LIN {X 0,Y 539.068,Z 532.449,A -85,B 0,C 180,E1 4627.318,E2 4627.318} C_VEL
LIN {X 0,Y 539.511,Z 496.056,A -85,B 0,C 180,E1 4628.109,E2 4628.109} C_VEL
LIN {X 0,Y 522.356,Z 463.143,A -85,B 0,C 180,E1 4630.176,E2 4630.176} C_VEL
LIN {X 0,Y 522.421,Z 462.44,A -85,B 0,C 180,E1 4635.931,E2 4635.931} C_VEL
LIN {X 0,Y 522.358,Z 462.44,A -85,B 0,C 180,E1 4641.503,E2 4641.503} C_VEL
LIN {X 0,Y 522.384,Z 462.44,A -85,B 0,C 180,E1 4647.2,E2 4647.2} C_VEL
LIN {X 0,Y 522.47,Z 462.44,A -85,B 0,C 180,E1 4652.377,E2 4652.377} C_VEL
LIN {X 0,Y 522.638,Z 462.44,A -85,B 0,C 180,E1 4657.983,E2 4657.983} C_VEL
LIN {X 0,Y 522.677,Z 462.44,A -85,B 0,C 180,E1 4663.162,E2 4663.162} C_VEL
LIN {X 0,Y 522.728,Z 462.44,A -85,B 0,C 180,E1 4670.012,E2 4670.012} C_VEL
LIN {X 0,Y 522.901,Z 462.44,A -85,B 0,C 180,E1 4675.016,E2 4675.016} C_VEL
LIN {X 0,Y 522.923,Z 462.44,A -85,B 0,C 180,E1 4679.999,E2 4679.999} C_VEL
LIN {X 0,Y 522.848,Z 462.44,A -85,B 0,C 180,E1 4684.982,E2 4684.982} C_VEL
LIN {X 0,Y 522.787,Z 462.44,A -85,B 0,C 180,E1 4690.024,E2 4690.024} C_VEL
LIN {X 0,Y 522.67,Z 462.44,A -85,B 0,C 180,E1 4695.11,E2 4695.11} C_VEL
LIN {X 0,Y 522.589,Z 462.44,A -85,B 0,C 180,E1 4700.342,E2 4700.342} C_VEL
LIN {X 0,Y 522.421,Z 462.44,A -85,B 0,C 180,E1 4706.042,E2 4706.042} C_VEL
LIN {X 0,Y 522.407,Z 462.44,A -85,B 0,C 180,E1 4711.442,E2 4711.442} C_VEL
LIN {X 0,Y 522.38,Z 462.44,A -85,B 0,C 180,E1 4717.488,E2 4717.488} C_VEL
LIN {X 0,Y 522.212,Z 462.44,A -85,B 0,C 180,E1 4723.542,E2 4723.542} C_VEL
LIN {X 0,Y 522.348,Z 462.44,A -85,B 0,C 180,E1 4728.899,E2 4728.899} C_VEL
LIN {X 0,Y 522.594,Z 462.44,A -85,B 0,C 180,E1 4734.992,E2 4734.992} C_VEL
LIN {X 0,Y 535.97,Z 492.125,A -85,B 0,C 180,E1 4736.47,E2 4736.47} C_VEL
LIN {X 0,Y 535.438,Z 535.67,A -85,B 0,C 180,E1 4737.354,E2 4737.354} C_VEL
LIN {X 0,Y 533.837,Z 572.448,A -85,B 0,C 180,E1 4738.666,E2 4738.666} C_VEL
LIN {X 0,Y 531.767,Z 608.408,A -85,B 0,C 180,E1 4740.582,E2 4740.582} C_VEL
LIN {X 0,Y 529.464,Z 642.826,A -85,B 0,C 180,E1 4743.115,E2 4743.115} C_VEL
LIN {X 0,Y 527.341,Z 673.183,A -85,B 0,C 180,E1 4746.073,E2 4746.073} C_VEL
LIN {X 0,Y 525.539,Z 700.097,A -85,B 0,C 180,E1 4749.484,E2 4749.484} C_VEL
LIN {X 0,Y 524.279,Z 723.704,A -85,B 0,C 180,E1 4753.43,E2 4753.43} C_VEL
LIN {X 0,Y 523.54,Z 741.491,A -85,B 0,C 180,E1 4757.473,E2 4757.473} C_VEL
LIN {X 0,Y 523.247,Z 754.217,A -85,B 0,C 180,E1 4761.681,E2 4761.681} C_VEL
LIN {X 0,Y 523.13,Z 760.5,A -85,B 0,C 180,E1 4765.019,E2 4765.019} C_VEL
LIN {X 0,Y 523.088,Z 763.612,A -85,B 0,C 180,E1 4768.341,E2 4768.341} C_VEL
LIN {X 0,Y 523.184,Z 763.555,A -85,B 0,C 180,E1 4771.658,E2 4771.658} C_VEL
LIN {X 0,Y 523.211,Z 759.15,A -85,B 0,C 180,E1 4775.813,E2 4775.813} C_VEL
LIN {X 0,Y 523.34,Z 749.587,A -85,B 0,C 180,E1 4779.997,E2 4779.997} C_VEL
LIN {X 0,Y 523.808,Z 734.142,A -85,B 0,C 180,E1 4784.287,E2 4784.287} C_VEL
LIN {X 0,Y 524.881,Z 712.493,A -85,B 0,C 180,E1 4788.501,E2 4788.501} C_VEL
LIN {X 0,Y 526.437,Z 686.433,A -85,B 0,C 180,E1 4792.268,E2 4792.268} C_VEL
LIN {X 0,Y 528.502,Z 656.362,A -85,B 0,C 180,E1 4795.571,E2 4795.571} C_VEL
LIN {X 0,Y 530.794,Z 623.032,A -85,B 0,C 180,E1 4798.343,E2 4798.343} C_VEL
LIN {X 0,Y 532.941,Z 589.022,A -85,B 0,C 180,E1 4800.442,E2 4800.442} C_VEL
LIN {X 0,Y 534.766,Z 553.339,A -85,B 0,C 180,E1 4802.003,E2 4802.003} C_VEL
LIN {X 0,Y 535.972,Z 516.697,A -85,B 0,C 180,E1 4803.016,E2 4803.016} C_VEL
LIN {X 0,Y 535.534,Z 491.051,A -85,B 0,C 180,E1 4803.488,E2 4803.488} C_VEL
LIN {X 0,Y 522.397,Z 462.44,A -85,B 0,C 180,E1 4805.02,E2 4805.02} C_VEL
LIN {X 0,Y 522.353,Z 462.44,A -85,B 0,C 180,E1 4811.101,E2 4811.101} C_VEL
LIN {X 0,Y 522.357,Z 462.44,A -85,B 0,C 180,E1 4816.441,E2 4816.441} C_VEL
LIN {X 0,Y 522.293,Z 462.44,A -85,B 0,C 180,E1 4822.504,E2 4822.504} C_VEL
LIN {X 0,Y 522.342,Z 462.44,A -85,B 0,C 180,E1 4828.554,E2 4828.554} C_VEL
LIN {X 0,Y 522.502,Z 462.44,A -85,B 0,C 180,E1 4834.24,E2 4834.24} C_VEL
LIN {X 0,Y 522.655,Z 462.44,A -85,B 0,C 180,E1 4839.66,E2 4839.66} C_VEL
LIN {X 0,Y 522.798,Z 462.44,A -85,B 0,C 180,E1 4844.894,E2 4844.894} C_VEL
LIN {X 0,Y 522.789,Z 462.44,A -85,B 0,C 180,E1 4851.23,E2 4851.23} C_VEL
LIN {X 0,Y 523.02,Z 462.44,A -85,B 0,C 180,E1 4856.682,E2 4856.682} C_VEL
LIN {X 0,Y 523.103,Z 462.44,A -85,B 0,C 180,E1 4861.659,E2 4861.659} C_VEL
LIN {X 0,Y 522.951,Z 462.44,A -85,B 0,C 180,E1 4866.651,E2 4866.651} C_VEL
LIN {X 0,Y 522.767,Z 462.44,A -85,B 0,C 180,E1 4871.697,E2 4871.697} C_VEL
LIN {X 0,Y 522.616,Z 462.44,A -85,B 0,C 180,E1 4877.043,E2 4877.043} C_VEL
LIN {X 0,Y 522.614,Z 462.44,A -85,B 0,C 180,E1 4882.124,E2 4882.124} C_VEL
LIN {X 0,Y 522.476,Z 462.44,A -85,B 0,C 180,E1 4887.622,E2 4887.622} C_VEL
LIN {X 0,Y 522.352,Z 462.44,A -85,B 0,C 180,E1 4892.514,E2 4892.514} C_VEL
LIN {X 0,Y 519.895,Z 462.44,A -85,B 0,C 180,E1 4893.928,E2 4893.928} C_VEL
LIN {X 0,Y 514.521,Z 462.44,A -85,B 0,C 180,E1 4896.046,E2 4896.046} C_VEL
LIN {X 0,Y 514.418,Z 462.44,A -85,B 0,C 180,E1 4896.292,E2 4896.292} C_VEL
LIN {X 0,Y 514.484,Z 462.44,A -85,B 0,C 180,E1 4902.629,E2 4902.629} C_VEL
LIN {X 0,Y 514.424,Z 462.947,A -85,B 0,C 180,E1 4909.174,E2 4909.174} C_VEL
LIN {X 0,Y 525.004,Z 483.039,A -85,B 0,C 180,E1 4910.412,E2 4910.412} C_VEL
LIN {X 0,Y 533.703,Z 501.5,A -85,B 0,C 180,E1 4911.496,E2 4911.496} C_VEL
LIN {X 0,Y 532.173,Z 544.934,A -85,B 0,C 180,E1 4912.524,E2 4912.524} C_VEL
LIN {X 0,Y 529.677,Z 588.035,A -85,B 0,C 180,E1 4914.292,E2 4914.292} C_VEL
LIN {X 0,Y 526.477,Z 629.276,A -85,B 0,C 180,E1 4916.773,E2 4916.773} C_VEL
LIN {X 0,Y 523.242,Z 667.514,A -85,B 0,C 180,E1 4919.932,E2 4919.932} C_VEL
LIN {X 0,Y 520.398,Z 700.092,A -85,B 0,C 180,E1 4923.454,E2 4923.454} C_VEL
LIN {X 0,Y 518.057,Z 730.026,A -85,B 0,C 180,E1 4927.669,E2 4927.669} C_VEL
LIN {X 0,Y 516.559,Z 753.744,A -85,B 0,C 180,E1 4932.054,E2 4932.054} C_VEL
LIN {X 0,Y 515.736,Z 772.742,A -85,B 0,C 180,E1 4936.848,E2 4936.848} C_VEL
LIN {X 0,Y 515.308,Z 785.33,A -85,B 0,C 180,E1 4941.552,E2 4941.552} C_VEL
LIN {X 0,Y 515.391,Z 790.904,A -85,B 0,C 180,E1 4944.944,E2 4944.944} C_VEL
LIN {X 0,Y 515.296,Z 793.657,A -85,B 0,C 180,E1 4948.316,E2 4948.316} C_VEL
LIN {X 0,Y 515.217,Z 792.628,A -85,B 0,C 180,E1 4953.37,E2 4953.37} C_VEL
LIN {X 0,Y 515.336,Z 786.917,A -85,B 0,C 180,E1 4957.598,E2 4957.598} C_VEL
LIN {X 0,Y 515.477,Z 776.771,A -85,B 0,C 180,E1 4961.865,E2 4961.865} C_VEL
LIN {X 0,Y 516.124,Z 761.488,A -85,B 0,C 180,E1 4966.182,E2 4966.182} C_VEL
LIN {X 0,Y 517.307,Z 740.375,A -85,B 0,C 180,E1 4970.563,E2 4970.563} C_VEL
LIN {X 0,Y 519.171,Z 714.818,A -85,B 0,C 180,E1 4974.608,E2 4974.608} C_VEL
LIN {X 0,Y 521.784,Z 684.177,A -85,B 0,C 180,E1 4978.371,E2 4978.371} C_VEL
LIN {X 0,Y 524.76,Z 650.107,A -85,B 0,C 180,E1 4981.614,E2 4981.614} C_VEL
LIN {X 0,Y 527.73,Z 614.196,A -85,B 0,C 180,E1 4984.231,E2 4984.231} C_VEL
LIN {X 0,Y 530.638,Z 574.086,A -85,B 0,C 180,E1 4986.362,E2 4986.362} C_VEL
LIN {X 0,Y 532.788,Z 532.447,A -85,B 0,C 180,E1 4987.835,E2 4987.835} C_VEL
LIN {X 0,Y 533.34,Z 499.06,A -85,B 0,C 180,E1 4988.58,E2 4988.58} C_VEL
LIN {X 0,Y 514.575,Z 464.052,A -85,B 0,C 180,E1 4990.795,E2 4990.795} C_VEL
LIN {X 0,Y 514.404,Z 462.44,A -85,B 0,C 180,E1 4990.993,E2 4990.993} C_VEL
LIN {X 0,Y 514.484,Z 462.44,A -85,B 0,C 180,E1 4997.404,E2 4997.404} C_VEL
LIN {X 0,Y 514.46,Z 462.44,A -85,B 0,C 180,E1 5002.622,E2 5002.622} C_VEL
LIN {X 0,Y 514.474,Z 462.44,A -85,B 0,C 180,E1 5008.593,E2 5008.593} C_VEL
LIN {X 0,Y 514.588,Z 462.44,A -85,B 0,C 180,E1 5013.811,E2 5013.811} C_VEL
LIN {X 0,Y 514.737,Z 462.44,A -85,B 0,C 180,E1 5020.271,E2 5020.271} C_VEL
LIN {X 0,Y 514.559,Z 462.44,A -85,B 0,C 180,E1 5026.181,E2 5026.181} C_VEL
LIN {X 0,Y 514.812,Z 462.44,A -85,B 0,C 180,E1 5031.544,E2 5031.544} C_VEL
LIN {X 0,Y 514.985,Z 462.44,A -85,B 0,C 180,E1 5036.628,E2 5036.628} C_VEL
LIN {X 0,Y 514.988,Z 462.44,A -85,B 0,C 180,E1 5041.684,E2 5041.684} C_VEL
LIN {X 0,Y 514.887,Z 462.44,A -85,B 0,C 180,E1 5046.753,E2 5046.753} C_VEL
LIN {X 0,Y 514.784,Z 462.44,A -85,B 0,C 180,E1 5051.879,E2 5051.879} C_VEL
LIN {X 0,Y 514.7,Z 462.44,A -85,B 0,C 180,E1 5057.105,E2 5057.105} C_VEL
LIN {X 0,Y 514.624,Z 462.44,A -85,B 0,C 180,E1 5062.484,E2 5062.484} C_VEL
LIN {X 0,Y 514.455,Z 462.44,A -85,B 0,C 180,E1 5068.089,E2 5068.089} C_VEL
LIN {X 0,Y 514.508,Z 462.44,A -85,B 0,C 180,E1 5073.991,E2 5073.991} C_VEL
LIN {X 0,Y 514.441,Z 462.44,A -85,B 0,C 180,E1 5080.071,E2 5080.071} C_VEL
LIN {X 0,Y 514.235,Z 462.44,A -85,B 0,C 180,E1 5085.036,E2 5085.036} C_VEL
LIN {X 0,Y 514.457,Z 462.44,A -85,B 0,C 180,E1 5089.917,E2 5089.917} C_VEL
LIN {X 0,Y 514.646,Z 462.711,A -85,B 0,C 180,E1 5094.315,E2 5094.315} C_VEL
LIN {X 0,Y 529.385,Z 494.183,A -85,B 0,C 180,E1 5096.03,E2 5096.03} C_VEL
LIN {X 0,Y 528.695,Z 537.141,A -85,B 0,C 180,E1 5096.931,E2 5096.931} C_VEL
LIN {X 0,Y 526.913,Z 574.501,A -85,B 0,C 180,E1 5098.31,E2 5098.31} C_VEL
LIN {X 0,Y 524.661,Z 609.82,A -85,B 0,C 180,E1 5100.243,E2 5100.243} C_VEL
LIN {X 0,Y 522.143,Z 644.081,A -85,B 0,C 180,E1 5102.824,E2 5102.824} C_VEL
LIN {X 0,Y 519.779,Z 675.099,A -85,B 0,C 180,E1 5105.932,E2 5105.932} C_VEL
LIN {X 0,Y 517.806,Z 702.022,A -85,B 0,C 180,E1 5109.458,E2 5109.458} C_VEL
LIN {X 0,Y 516.471,Z 724.789,A -85,B 0,C 180,E1 5113.391,E2 5113.391} C_VEL
LIN {X 0,Y 515.709,Z 741.489,A -85,B 0,C 180,E1 5117.279,E2 5117.279} C_VEL
LIN {X 0,Y 515.361,Z 754.215,A -85,B 0,C 180,E1 5121.553,E2 5121.553} C_VEL
LIN {X 0,Y 515.251,Z 760.499,A -85,B 0,C 180,E1 5124.942,E2 5124.942} C_VEL
LIN {X 0,Y 515.185,Z 763.612,A -85,B 0,C 180,E1 5128.316,E2 5128.316} C_VEL
LIN {X 0,Y 515.201,Z 763.101,A -85,B 0,C 180,E1 5132.437,E2 5132.437} C_VEL
LIN {X 0,Y 515.309,Z 757.598,A -85,B 0,C 180,E1 5136.75,E2 5136.75} C_VEL
LIN {X 0,Y 515.502,Z 748.281,A -85,B 0,C 180,E1 5140.589,E2 5140.589} C_VEL
LIN {X 0,Y 516.085,Z 732.756,A -85,B 0,C 180,E1 5144.82,E2 5144.82} C_VEL
LIN {X 0,Y 517.301,Z 711.169,A -85,B 0,C 180,E1 5149.004,E2 5149.004} C_VEL
LIN {X 0,Y 518.994,Z 685.739,A -85,B 0,C 180,E1 5152.695,E2 5152.695} C_VEL
LIN {X 0,Y 521.168,Z 656.428,A -85,B 0,C 180,E1 5155.951,E2 5155.951} C_VEL
LIN {X 0,Y 523.723,Z 622.883,A -85,B 0,C 180,E1 5158.773,E2 5158.773} C_VEL
LIN {X 0,Y 526.138,Z 587.932,A -85,B 0,C 180,E1 5160.941,E2 5160.941} C_VEL
LIN {X 0,Y 528.053,Z 552.594,A -85,B 0,C 180,E1 5162.487,E2 5162.487} C_VEL
LIN {X 0,Y 529.405,Z 513.93,A -85,B 0,C 180,E1 5163.533,E2 5163.533} C_VEL
LIN {X 0,Y 529.025,Z 493.82,A -85,B 0,C 180,E1 5163.912,E2 5163.912} C_VEL
LIN {X 0,Y 514.476,Z 462.44,A -85,B 0,C 180,E1 5165.67,E2 5165.67} C_VEL
LIN {X 0,Y 514.446,Z 462.44,A -85,B 0,C 180,E1 5170.354,E2 5170.354} C_VEL
LIN {X 0,Y 514.346,Z 462.44,A -85,B 0,C 180,E1 5175.056,E2 5175.056} C_VEL
LIN {X 0,Y 514.413,Z 462.44,A -85,B 0,C 180,E1 5179.933,E2 5179.933} C_VEL
LIN {X 0,Y 514.37,Z 462.44,A -85,B 0,C 180,E1 5185.999,E2 5185.999} C_VEL
LIN {X 0,Y 514.517,Z 462.44,A -85,B 0,C 180,E1 5191.988,E2 5191.988} C_VEL
LIN {X 0,Y 514.658,Z 462.44,A -85,B 0,C 180,E1 5197.518,E2 5197.518} C_VEL
LIN {X 0,Y 514.802,Z 462.44,A -85,B 0,C 180,E1 5202.898,E2 5202.898} C_VEL
LIN {X 0,Y 514.854,Z 462.44,A -85,B 0,C 180,E1 5208.122,E2 5208.122} C_VEL
LIN {X 0,Y 514.886,Z 462.44,A -85,B 0,C 180,E1 5213.247,E2 5213.247} C_VEL
LIN {X 0,Y 514.978,Z 462.44,A -85,B 0,C 180,E1 5218.522,E2 5218.522} C_VEL
LIN {X 0,Y 514.986,Z 462.44,A -85,B 0,C 180,E1 5223.372,E2 5223.372} C_VEL
LIN {X 0,Y 514.833,Z 462.44,A -85,B 0,C 180,E1 5228.456,E2 5228.456} C_VEL
LIN {X 0,Y 514.77,Z 462.44,A -85,B 0,C 180,E1 5233.914,E2 5233.914} C_VEL
LIN {X 0,Y 514.643,Z 462.44,A -85,B 0,C 180,E1 5239.699,E2 5239.699} C_VEL
LIN {X 0,Y 514.658,Z 462.44,A -85,B 0,C 180,E1 5244.321,E2 5244.321} C_VEL
LIN {X 0,Y 514.452,Z 462.44,A -85,B 0,C 180,E1 5250.02,E2 5250.02} C_VEL
LIN {X 0,Y 514.418,Z 462.44,A -85,B 0,C 180,E1 5256.292,E2 5256.292} C_VEL
LIN {X 0,Y 513.127,Z 462.44,A -85,B 0,C 180,E1 5257.254,E2 5257.254} C_VEL
LIN {X 0,Y 506.498,Z 462.44,A -85,B 0,C 180,E1 5259.877,E2 5259.877} C_VEL
LIN {X 0,Y 506.409,Z 462.44,A -85,B 0,C 180,E1 5260.126,E2 5260.126} C_VEL
LIN {X 0,Y 506.426,Z 462.44,A -85,B 0,C 180,E1 5265.848,E2 5265.848} C_VEL
LIN {X 0,Y 506.519,Z 462.44,A -85,B 0,C 180,E1 5268.469,E2 5268.469} C_VEL
LIN {X 0,Y 513.608,Z 477.407,A -85,B 0,C 180,E1 5269.354,E2 5269.354} C_VEL
LIN {X 0,Y 527.461,Z 502.782,A -85,B 0,C 180,E1 5270.981,E2 5270.981} C_VEL
LIN {X 0,Y 525.883,Z 544.972,A -85,B 0,C 180,E1 5271.999,E2 5271.999} C_VEL
LIN {X 0,Y 523.263,Z 586.974,A -85,B 0,C 180,E1 5273.727,E2 5273.727} C_VEL
LIN {X 0,Y 520.006,Z 626.15,A -85,B 0,C 180,E1 5276.067,E2 5276.067} C_VEL
LIN {X 0,Y 516.604,Z 662.655,A -85,B 0,C 180,E1 5279.019,E2 5279.019} C_VEL
LIN {X 0,Y 513.42,Z 695.798,A -85,B 0,C 180,E1 5282.526,E2 5282.526} C_VEL
LIN {X 0,Y 510.94,Z 724.214,A -85,B 0,C 180,E1 5286.4,E2 5286.4} C_VEL
LIN {X 0,Y 509.104,Z 747.619,A -85,B 0,C 180,E1 5290.497,E2 5290.497} C_VEL
LIN {X 0,Y 508.049,Z 766.783,A -85,B 0,C 180,E1 5294.914,E2 5294.914} C_VEL
LIN {X 0,Y 507.515,Z 781.436,A -85,B 0,C 180,E1 5299.688,E2 5299.688} C_VEL
LIN {X 0,Y 507.411,Z 789.703,A -85,B 0,C 180,E1 5304.005,E2 5304.005} C_VEL
LIN {X 0,Y 507.409,Z 793.657,A -85,B 0,C 180,E1 5308.29,E2 5308.29} C_VEL
LIN {X 0,Y 507.322,Z 793.657,A -85,B 0,C 180,E1 5311.71,E2 5311.71} C_VEL
LIN {X 0,Y 507.437,Z 788.478,A -85,B 0,C 180,E1 5316.855,E2 5316.855} C_VEL
LIN {X 0,Y 507.61,Z 777.986,A -85,B 0,C 180,E1 5321.616,E2 5321.616} C_VEL
LIN {X 0,Y 508.238,Z 763.242,A -85,B 0,C 180,E1 5325.996,E2 5325.996} C_VEL
LIN {X 0,Y 509.47,Z 743.034,A -85,B 0,C 180,E1 5330.391,E2 5330.391} C_VEL
LIN {X 0,Y 511.491,Z 717.337,A -85,B 0,C 180,E1 5334.635,E2 5334.635} C_VEL
LIN {X 0,Y 514.386,Z 686.273,A -85,B 0,C 180,E1 5338.576,E2 5338.576} C_VEL
LIN {X 0,Y 517.734,Z 651.136,A -85,B 0,C 180,E1 5342.002,E2 5342.002} C_VEL
LIN {X 0,Y 521.129,Z 613.628,A -85,B 0,C 180,E1 5344.764,E2 5344.764} C_VEL
LIN {X 0,Y 524.221,Z 573.752,A -85,B 0,C 180,E1 5346.897,E2 5346.897} C_VEL
LIN {X 0,Y 526.537,Z 532.365,A -85,B 0,C 180,E1 5348.367,E2 5348.367} C_VEL
LIN {X 0,Y 526.984,Z 501.734,A -85,B 0,C 180,E1 5349.083,E2 5349.083} C_VEL
LIN {X 0,Y 506.577,Z 463.424,A -85,B 0,C 180,E1 5351.481,E2 5351.481} C_VEL
LIN {X 0,Y 506.528,Z 462.44,A -85,B 0,C 180,E1 5351.649,E2 5351.649} C_VEL
LIN {X 0,Y 506.513,Z 462.44,A -85,B 0,C 180,E1 5358.36,E2 5358.36} C_VEL
LIN {X 0,Y 506.542,Z 462.44,A -85,B 0,C 180,E1 5363.811,E2 5363.811} C_VEL
LIN {X 0,Y 506.542,Z 462.44,A -85,B 0,C 180,E1 5370.095,E2 5370.095} C_VEL
LIN {X 0,Y 506.688,Z 462.44,A -85,B 0,C 180,E1 5375.271,E2 5375.271} C_VEL
LIN {X 0,Y 506.863,Z 462.44,A -85,B 0,C 180,E1 5380.818,E2 5380.818} C_VEL
LIN {X 0,Y 506.673,Z 462.44,A -85,B 0,C 180,E1 5386.169,E2 5386.169} C_VEL
LIN {X 0,Y 506.895,Z 462.44,A -85,B 0,C 180,E1 5391.411,E2 5391.411} C_VEL
LIN {X 0,Y 507.079,Z 462.44,A -85,B 0,C 180,E1 5396.576,E2 5396.576} C_VEL
LIN {X 0,Y 507.087,Z 462.44,A -85,B 0,C 180,E1 5401.71,E2 5401.71} C_VEL
LIN {X 0,Y 506.976,Z 462.44,A -85,B 0,C 180,E1 5406.859,E2 5406.859} C_VEL
LIN {X 0,Y 506.864,Z 462.44,A -85,B 0,C 180,E1 5412.068,E2 5412.068} C_VEL
LIN {X 0,Y 506.792,Z 462.44,A -85,B 0,C 180,E1 5417.38,E2 5417.38} C_VEL
LIN {X 0,Y 506.708,Z 462.44,A -85,B 0,C 180,E1 5422.855,E2 5422.855} C_VEL
LIN {X 0,Y 506.505,Z 462.44,A -85,B 0,C 180,E1 5428.57,E2 5428.57} C_VEL
LIN {X 0,Y 506.594,Z 462.44,A -85,B 0,C 180,E1 5434.597,E2 5434.597} C_VEL
LIN {X 0,Y 506.406,Z 462.44,A -85,B 0,C 180,E1 5441.124,E2 5441.124} C_VEL
LIN {X 0,Y 506.291,Z 462.44,A -85,B 0,C 180,E1 5446.54,E2 5446.54} C_VEL
LIN {X 0,Y 506.637,Z 462.44,A -85,B 0,C 180,E1 5453.293,E2 5453.293} C_VEL
LIN {X 0,Y 506.699,Z 463.166,A -85,B 0,C 180,E1 5453.568,E2 5453.568} C_VEL
LIN {X 0,Y 522.828,Z 496.797,A -85,B 0,C 180,E1 5455.588,E2 5455.588} C_VEL
LIN {X 0,Y 521.989,Z 538.781,A -85,B 0,C 180,E1 5456.503,E2 5456.503} C_VEL
LIN {X 0,Y 520.049,Z 575.663,A -85,B 0,C 180,E1 5457.901,E2 5457.901} C_VEL
LIN {X 0,Y 517.555,Z 611.609,A -85,B 0,C 180,E1 5459.92,E2 5459.92} C_VEL
LIN {X 0,Y 514.849,Z 645.336,A -85,B 0,C 180,E1 5462.525,E2 5462.525} C_VEL
LIN {X 0,Y 512.257,Z 676.316,A -85,B 0,C 180,E1 5465.703,E2 5465.703} C_VEL
LIN {X 0,Y 510.082,Z 703.485,A -85,B 0,C 180,E1 5469.361,E2 5469.361} C_VEL
LIN {X 0,Y 508.671,Z 725.871,A -85,B 0,C 180,E1 5473.351,E2 5473.351} C_VEL
LIN {X 0,Y 507.779,Z 743.023,A -85,B 0,C 180,E1 5477.515,E2 5477.515} C_VEL
LIN {X 0,Y 507.478,Z 754.214,A -85,B 0,C 180,E1 5481.42,E2 5481.42} C_VEL
LIN {X 0,Y 507.354,Z 760.498,A -85,B 0,C 180,E1 5484.863,E2 5484.863} C_VEL
LIN {X 0,Y 507.306,Z 763.611,A -85,B 0,C 180,E1 5488.29,E2 5488.29} C_VEL
LIN {X 0,Y 507.393,Z 763.556,A -85,B 0,C 180,E1 5491.71,E2 5491.71} C_VEL
LIN {X 0,Y 507.418,Z 759.153,A -85,B 0,C 180,E1 5495.995,E2 5495.995} C_VEL
LIN {X 0,Y 507.618,Z 749.591,A -85,B 0,C 180,E1 5500.31,E2 5500.31} C_VEL
LIN {X 0,Y 508.214,Z 734.209,A -85,B 0,C 180,E1 5504.72,E2 5504.72} C_VEL
LIN {X 0,Y 509.547,Z 712.499,A -85,B 0,C 180,E1 5509.079,E2 5509.079} C_VEL
LIN {X 0,Y 511.399,Z 687.196,A -85,B 0,C 180,E1 5512.86,E2 5512.86} C_VEL
LIN {X 0,Y 513.78,Z 657.585,A -85,B 0,C 180,E1 5516.235,E2 5516.235} C_VEL
LIN {X 0,Y 516.53,Z 624.859,A -85,B 0,C 180,E1 5519.058,E2 5519.058} C_VEL
LIN {X 0,Y 519.173,Z 589.613,A -85,B 0,C 180,E1 5521.307,E2 5521.307} C_VEL
LIN {X 0,Y 521.339,Z 553.567,A -85,B 0,C 180,E1 5522.922,E2 5522.922} C_VEL
LIN {X 0,Y 522.812,Z 514.592,A -85,B 0,C 180,E1 5524.001,E2 5524.001} C_VEL
LIN {X 0,Y 522.58,Z 496.624,A -85,B 0,C 180,E1 5524.343,E2 5524.343} C_VEL
LIN {X 0,Y 508.222,Z 467.264,A -85,B 0,C 180,E1 5526.119,E2 5526.119} C_VEL
LIN {X 0,Y 506.547,Z 462.44,A -85,B 0,C 180,E1 5526.428,E2 5526.428} C_VEL
LIN {X 0,Y 506.418,Z 462.44,A -85,B 0,C 180,E1 5531.637,E2 5531.637} C_VEL
LIN {X 0,Y 506.434,Z 462.44,A -85,B 0,C 180,E1 5538.37,E2 5538.37} C_VEL
LIN {X 0,Y 506.499,Z 462.44,A -85,B 0,C 180,E1 5543.818,E2 5543.818} C_VEL
LIN {X 0,Y 506.542,Z 462.44,A -85,B 0,C 180,E1 5550.096,E2 5550.096} C_VEL
LIN {X 0,Y 506.66,Z 462.44,A -85,B 0,C 180,E1 5555.272,E2 5555.272} C_VEL
LIN {X 0,Y 506.846,Z 462.44,A -85,B 0,C 180,E1 5560.819,E2 5560.819} C_VEL
LIN {X 0,Y 507.006,Z 462.44,A -85,B 0,C 180,E1 5566.18,E2 5566.18} C_VEL
LIN {X 0,Y 507.031,Z 462.44,A -85,B 0,C 180,E1 5571.415,E2 5571.415} C_VEL
LIN {X 0,Y 507.201,Z 462.44,A -85,B 0,C 180,E1 5576.578,E2 5576.578} C_VEL
LIN {X 0,Y 507.319,Z 462.44,A -85,B 0,C 180,E1 5581.711,E2 5581.711} C_VEL
LIN {X 0,Y 507.112,Z 462.44,A -85,B 0,C 180,E1 5586.859,E2 5586.859} C_VEL
LIN {X 0,Y 506.908,Z 462.44,A -85,B 0,C 180,E1 5592.069,E2 5592.069} C_VEL
LIN {X 0,Y 506.801,Z 462.44,A -85,B 0,C 180,E1 5597.382,E2 5597.382} C_VEL
LIN {X 0,Y 506.753,Z 462.44,A -85,B 0,C 180,E1 5602.855,E2 5602.855} C_VEL
LIN {X 0,Y 506.55,Z 462.44,A -85,B 0,C 180,E1 5608.569,E2 5608.569} C_VEL
LIN {X 0,Y 506.491,Z 462.44,A -85,B 0,C 180,E1 5614.607,E2 5614.607} C_VEL
LIN {X 0,Y 506.409,Z 462.44,A -85,B 0,C 180,E1 5620.126,E2 5620.126} C_VEL
LIN {X 0,Y 503.917,Z 462.44,A -85,B 0,C 180,E1 5621.586,E2 5621.586} C_VEL
LIN {X 0,Y 498.644,Z 462.44,A -85,B 0,C 180,E1 5623.776,E2 5623.776} C_VEL
LIN {X 0,Y 498.557,Z 462.44,A -85,B 0,C 180,E1 5624.029,E2 5624.029} C_VEL
LIN {X 0,Y 498.543,Z 462.44,A -85,B 0,C 180,E1 5627.772,E2 5627.772} C_VEL
LIN {X 0,Y 508.311,Z 482.341,A -85,B 0,C 180,E1 5628.999,E2 5628.999} C_VEL
LIN {X 0,Y 521.269,Z 505.738,A -85,B 0,C 180,E1 5630.489,E2 5630.489} C_VEL
LIN {X 0,Y 519.525,Z 546.504,A -85,B 0,C 180,E1 5631.511,E2 5631.511} C_VEL
LIN {X 0,Y 516.701,Z 588.195,A -85,B 0,C 180,E1 5633.261,E2 5633.261} C_VEL
LIN {X 0,Y 513.105,Z 628.263,A -85,B 0,C 180,E1 5635.708,E2 5635.708} C_VEL
LIN {X 0,Y 509.277,Z 666.433,A -85,B 0,C 180,E1 5638.902,E2 5638.902} C_VEL
LIN {X 0,Y 505.8,Z 699.826,A -85,B 0,C 180,E1 5642.588,E2 5642.588} C_VEL
LIN {X 0,Y 502.86,Z 730.03,A -85,B 0,C 180,E1 5646.956,E2 5646.956} C_VEL
LIN {X 0,Y 501.012,Z 754.292,A -85,B 0,C 180,E1 5651.603,E2 5651.603} C_VEL
LIN {X 0,Y 500.037,Z 772.744,A -85,B 0,C 180,E1 5656.428,E2 5656.428} C_VEL
LIN {X 0,Y 499.528,Z 785.33,A -85,B 0,C 180,E1 5661.283,E2 5661.283} C_VEL
LIN {X 0,Y 499.575,Z 790.904,A -85,B 0,C 180,E1 5664.783,E2 5664.783} C_VEL
LIN {X 0,Y 499.507,Z 793.657,A -85,B 0,C 180,E1 5668.263,E2 5668.263} C_VEL
LIN {X 0,Y 499.42,Z 793.657,A -85,B 0,C 180,E1 5671.737,E2 5671.737} C_VEL
LIN {X 0,Y 499.513,Z 789.703,A -85,B 0,C 180,E1 5676.09,E2 5676.09} C_VEL
LIN {X 0,Y 499.737,Z 781.436,A -85,B 0,C 180,E1 5680.474,E2 5680.474} C_VEL
LIN {X 0,Y 500.299,Z 766.477,A -85,B 0,C 180,E1 5685.413,E2 5685.413} C_VEL
LIN {X 0,Y 501.525,Z 746.398,A -85,B 0,C 180,E1 5690.065,E2 5690.065} C_VEL
LIN {X 0,Y 503.756,Z 720.466,A -85,B 0,C 180,E1 5694.561,E2 5694.561} C_VEL
LIN {X 0,Y 506.992,Z 688.518,A -85,B 0,C 180,E1 5698.77,E2 5698.77} C_VEL
LIN {X 0,Y 510.71,Z 652.467,A -85,B 0,C 180,E1 5702.374,E2 5702.374} C_VEL
LIN {X 0,Y 514.349,Z 615.494,A -85,B 0,C 180,E1 5705.16,E2 5705.16} C_VEL
LIN {X 0,Y 517.72,Z 575.169,A -85,B 0,C 180,E1 5707.363,E2 5707.363} C_VEL
LIN {X 0,Y 520.24,Z 533.982,A -85,B 0,C 180,E1 5708.864,E2 5708.864} C_VEL
LIN {X 0,Y 520.88,Z 504.831,A -85,B 0,C 180,E1 5709.566,E2 5709.566} C_VEL
LIN {X 0,Y 498.635,Z 463.583,A -85,B 0,C 180,E1 5712.177,E2 5712.177} C_VEL
LIN {X 0,Y 498.554,Z 462.44,A -85,B 0,C 180,E1 5712.23,E2 5712.23} C_VEL
LIN {X 0,Y 498.578,Z 462.44,A -85,B 0,C 180,E1 5718.083,E2 5718.083} C_VEL
LIN {X 0,Y 498.574,Z 462.44,A -85,B 0,C 180,E1 5724.763,E2 5724.763} C_VEL
LIN {X 0,Y 498.616,Z 462.44,A -85,B 0,C 180,E1 5730.933,E2 5730.933} C_VEL
LIN {X 0,Y 498.786,Z 462.44,A -85,B 0,C 180,E1 5736.759,E2 5736.759} C_VEL
LIN {X 0,Y 498.917,Z 462.44,A -85,B 0,C 180,E1 5742.334,E2 5742.334} C_VEL
LIN {X 0,Y 498.821,Z 462.44,A -85,B 0,C 180,E1 5747.733,E2 5747.733} C_VEL
LIN {X 0,Y 499.182,Z 462.44,A -85,B 0,C 180,E1 5753.031,E2 5753.031} C_VEL
LIN {X 0,Y 499.43,Z 462.44,A -85,B 0,C 180,E1 5758.262,E2 5758.262} C_VEL
LIN {X 0,Y 499.274,Z 462.44,A -85,B 0,C 180,E1 5763.476,E2 5763.476} C_VEL
LIN {X 0,Y 499.093,Z 462.44,A -85,B 0,C 180,E1 5768.723,E2 5768.723} C_VEL
LIN {X 0,Y 498.971,Z 462.44,A -85,B 0,C 180,E1 5774.047,E2 5774.047} C_VEL
LIN {X 0,Y 498.811,Z 462.44,A -85,B 0,C 180,E1 5779.78,E2 5779.78} C_VEL
LIN {X 0,Y 498.702,Z 462.44,A -85,B 0,C 180,E1 5785.15,E2 5785.15} C_VEL
LIN {X 0,Y 498.612,Z 462.44,A -85,B 0,C 180,E1 5791.758,E2 5791.758} C_VEL
LIN {X 0,Y 498.548,Z 462.44,A -85,B 0,C 180,E1 5797.848,E2 5797.848} C_VEL
LIN {X 0,Y 498.366,Z 462.44,A -85,B 0,C 180,E1 5804.321,E2 5804.321} C_VEL
LIN {X 0,Y 498.524,Z 462.44,A -85,B 0,C 180,E1 5810.371,E2 5810.371} C_VEL
LIN {X 0,Y 498.64,Z 462.44,A -85,B 0,C 180,E1 5812.724,E2 5812.724} C_VEL
LIN {X 0,Y 501.28,Z 468.278,A -85,B 0,C 180,E1 5813.123,E2 5813.123} C_VEL
LIN {X 0,Y 516.271,Z 498.987,A -85,B 0,C 180,E1 5815.101,E2 5815.101} C_VEL
LIN {X 0,Y 515.141,Z 544.259,A -85,B 0,C 180,E1 5816.181,E2 5816.181} C_VEL
LIN {X 0,Y 512.794,Z 583.475,A -85,B 0,C 180,E1 5817.81,E2 5817.81} C_VEL
LIN {X 0,Y 509.917,Z 620.008,A -85,B 0,C 180,E1 5820.051,E2 5820.051} C_VEL
LIN {X 0,Y 506.905,Z 653.852,A -85,B 0,C 180,E1 5822.902,E2 5822.902} C_VEL
LIN {X 0,Y 504.079,Z 684.465,A -85,B 0,C 180,E1 5826.333,E2 5826.333} C_VEL
LIN {X 0,Y 501.915,Z 710.749,A -85,B 0,C 180,E1 5830.226,E2 5830.226} C_VEL
LIN {X 0,Y 500.581,Z 730.954,A -85,B 0,C 180,E1 5834.203,E2 5834.203} C_VEL
LIN {X 0,Y 499.831,Z 745.914,A -85,B 0,C 180,E1 5838.201,E2 5838.201} C_VEL
LIN {X 0,Y 499.576,Z 756.136,A -85,B 0,C 180,E1 5842.161,E2 5842.161} C_VEL
LIN {X 0,Y 499.394,Z 762.443,A -85,B 0,C 180,E1 5846.524,E2 5846.524} C_VEL
LIN {X 0,Y 499.433,Z 763.995,A -85,B 0,C 180,E1 5850,E2 5850} C_VEL
LIN {X 0,Y 499.421,Z 762.354,A -85,B 0,C 180,E1 5853.476,E2 5853.476} C_VEL
LIN {X 0,Y 499.617,Z 755.94,A -85,B 0,C 180,E1 5857.838,E2 5857.838} C_VEL
LIN {X 0,Y 499.991,Z 744.241,A -85,B 0,C 180,E1 5862.239,E2 5862.239} C_VEL
LIN {X 0,Y 500.895,Z 726.518,A -85,B 0,C 180,E1 5866.689,E2 5866.689} C_VEL
LIN {X 0,Y 502.449,Z 704.042,A -85,B 0,C 180,E1 5870.788,E2 5870.788} C_VEL
LIN {X 0,Y 504.817,Z 676.33,A -85,B 0,C 180,E1 5874.585,E2 5874.585} C_VEL
LIN {X 0,Y 507.658,Z 645.641,A -85,B 0,C 180,E1 5877.777,E2 5877.777} C_VEL
LIN {X 0,Y 510.505,Z 611.995,A -85,B 0,C 180,E1 5880.42,E2 5880.42} C_VEL
LIN {X 0,Y 513.222,Z 575.237,A -85,B 0,C 180,E1 5882.509,E2 5882.509} C_VEL
LIN {X 0,Y 515.443,Z 536.397,A -85,B 0,C 180,E1 5883.966,E2 5883.966} C_VEL
LIN {X 0,Y 516.246,Z 499.445,A -85,B 0,C 180,E1 5884.803,E2 5884.803} C_VEL
LIN {X 0,Y 501.063,Z 468.099,A -85,B 0,C 180,E1 5886.801,E2 5886.801} C_VEL
LIN {X 0,Y 498.573,Z 462.44,A -85,B 0,C 180,E1 5887.222,E2 5887.222} C_VEL
LIN {X 0,Y 498.482,Z 462.44,A -85,B 0,C 180,E1 5893.206,E2 5893.206} C_VEL
LIN {X 0,Y 498.453,Z 462.44,A -85,B 0,C 180,E1 5899.413,E2 5899.413} C_VEL
LIN {X 0,Y 498.544,Z 462.44,A -85,B 0,C 180,E1 5905.087,E2 5905.087} C_VEL
LIN {X 0,Y 498.615,Z 462.44,A -85,B 0,C 180,E1 5911.72,E2 5911.72} C_VEL
LIN {X 0,Y 498.774,Z 462.44,A -85,B 0,C 180,E1 5916.76,E2 5916.76} C_VEL
LIN {X 0,Y 498.928,Z 462.44,A -85,B 0,C 180,E1 5922.337,E2 5922.337} C_VEL
LIN {X 0,Y 499.022,Z 462.44,A -85,B 0,C 180,E1 5927.74,E2 5927.74} C_VEL
LIN {X 0,Y 499.069,Z 462.44,A -85,B 0,C 180,E1 5933.031,E2 5933.031} C_VEL
LIN {X 0,Y 499.203,Z 462.44,A -85,B 0,C 180,E1 5938.263,E2 5938.263} C_VEL
LIN {X 0,Y 499.176,Z 462.44,A -85,B 0,C 180,E1 5943.479,E2 5943.479} C_VEL
LIN {X 0,Y 499.032,Z 462.44,A -85,B 0,C 180,E1 5948.726,E2 5948.726} C_VEL
LIN {X 0,Y 498.972,Z 462.44,A -85,B 0,C 180,E1 5954.049,E2 5954.049} C_VEL
LIN {X 0,Y 498.801,Z 462.44,A -85,B 0,C 180,E1 5959.776,E2 5959.776} C_VEL
LIN {X 0,Y 498.776,Z 462.44,A -85,B 0,C 180,E1 5965.148,E2 5965.148} C_VEL
LIN {X 0,Y 498.546,Z 462.44,A -85,B 0,C 180,E1 5971.746,E2 5971.746} C_VEL
LIN {X 0,Y 498.537,Z 462.44,A -85,B 0,C 180,E1 5977.846,E2 5977.846} C_VEL
LIN {X 0,Y 498.557,Z 462.44,A -85,B 0,C 180,E1 5984.029,E2 5984.029} C_VEL
LIN {X 0,Y 494.571,Z 462.44,A -85,B 0,C 180,E1 5985.311,E2 5985.311} C_VEL
LIN {X 0,Y 490.63,Z 462.44,A -85,B 0,C 180,E1 5986.615,E2 5986.615} C_VEL
LIN {X 0,Y 490.676,Z 463.172,A -85,B 0,C 180,E1 5987.105,E2 5987.105} C_VEL
LIN {X 0,Y 514.876,Z 509.543,A -85,B 0,C 180,E1 5990.028,E2 5990.028} C_VEL
LIN {X 0,Y 513.105,Z 549.318,A -85,B 0,C 180,E1 5991.057,E2 5991.057} C_VEL
LIN {X 0,Y 510.152,Z 589.505,A -85,B 0,C 180,E1 5992.792,E2 5992.792} C_VEL
LIN {X 0,Y 506.285,Z 629.424,A -85,B 0,C 180,E1 5995.277,E2 5995.277} C_VEL
LIN {X 0,Y 502.201,Z 666.751,A -85,B 0,C 180,E1 5998.449,E2 5998.449} C_VEL
LIN {X 0,Y 498.406,Z 700.567,A -85,B 0,C 180,E1 6002.25,E2 6002.25} C_VEL
LIN {X 0,Y 495.331,Z 730.031,A -85,B 0,C 180,E1 6006.585,E2 6006.585} C_VEL
LIN {X 0,Y 493.311,Z 753.842,A -85,B 0,C 180,E1 6011.199,E2 6011.199} C_VEL
LIN {X 0,Y 492.198,Z 772.745,A -85,B 0,C 180,E1 6016.207,E2 6016.207} C_VEL
LIN {X 0,Y 491.647,Z 785.33,A -85,B 0,C 180,E1 6021.142,E2 6021.142} C_VEL
LIN {X 0,Y 491.665,Z 790.904,A -85,B 0,C 180,E1 6024.699,E2 6024.699} C_VEL
LIN {X 0,Y 491.602,Z 793.657,A -85,B 0,C 180,E1 6028.235,E2 6028.235} C_VEL
LIN {X 0,Y 491.516,Z 793.657,A -85,B 0,C 180,E1 6031.765,E2 6031.765} C_VEL
LIN {X 0,Y 491.634,Z 789.703,A -85,B 0,C 180,E1 6036.188,E2 6036.188} C_VEL
LIN {X 0,Y 491.856,Z 781.435,A -85,B 0,C 180,E1 6040.644,E2 6040.644} C_VEL
LIN {X 0,Y 492.469,Z 766.677,A -85,B 0,C 180,E1 6045.606,E2 6045.606} C_VEL
LIN {X 0,Y 493.812,Z 746.746,A -85,B 0,C 180,E1 6050.318,E2 6050.318} C_VEL
LIN {X 0,Y 496.173,Z 721.693,A -85,B 0,C 180,E1 6054.761,E2 6054.761} C_VEL
LIN {X 0,Y 499.393,Z 692.012,A -85,B 0,C 180,E1 6058.802,E2 6058.802} C_VEL
LIN {X 0,Y 503.161,Z 658.338,A -85,B 0,C 180,E1 6062.339,E2 6062.339} C_VEL
LIN {X 0,Y 506.98,Z 622.299,A -85,B 0,C 180,E1 6065.225,E2 6065.225} C_VEL
LIN {X 0,Y 510.592,Z 583.865,A -85,B 0,C 180,E1 6067.495,E2 6067.495} C_VEL
LIN {X 0,Y 513.415,Z 543.22,A -85,B 0,C 180,E1 6069.152,E2 6069.152} C_VEL
LIN {X 0,Y 514.67,Z 508.009,A -85,B 0,C 180,E1 6070.019,E2 6070.019} C_VEL
LIN {X 0,Y 490.719,Z 463.658,A -85,B 0,C 180,E1 6072.9,E2 6072.9} C_VEL
LIN {X 0,Y 490.639,Z 462.44,A -85,B 0,C 180,E1 6073.091,E2 6073.091} C_VEL
LIN {X 0,Y 490.621,Z 462.44,A -85,B 0,C 180,E1 6079.607,E2 6079.607} C_VEL
LIN {X 0,Y 490.624,Z 462.44,A -85,B 0,C 180,E1 6086.258,E2 6086.258} C_VEL
LIN {X 0,Y 490.725,Z 462.44,A -85,B 0,C 180,E1 6092.433,E2 6092.433} C_VEL
LIN {X 0,Y 490.901,Z 462.44,A -85,B 0,C 180,E1 6098.278,E2 6098.278} C_VEL
LIN {X 0,Y 490.92,Z 462.44,A -85,B 0,C 180,E1 6103.885,E2 6103.885} C_VEL
LIN {X 0,Y 491.032,Z 462.44,A -85,B 0,C 180,E1 6110.661,E2 6110.661} C_VEL
LIN {X 0,Y 491.269,Z 462.44,A -85,B 0,C 180,E1 6116.465,E2 6116.465} C_VEL
LIN {X 0,Y 491.3,Z 462.44,A -85,B 0,C 180,E1 6121.765,E2 6121.765} C_VEL
LIN {X 0,Y 491.153,Z 462.44,A -85,B 0,C 180,E1 6127.081,E2 6127.081} C_VEL
LIN {X 0,Y 491.036,Z 462.44,A -85,B 0,C 180,E1 6132.463,E2 6132.463} C_VEL
LIN {X 0,Y 490.941,Z 462.44,A -85,B 0,C 180,E1 6137.96,E2 6137.96} C_VEL
LIN {X 0,Y 490.814,Z 462.44,A -85,B 0,C 180,E1 6143.639,E2 6143.639} C_VEL
LIN {X 0,Y 490.646,Z 462.44,A -85,B 0,C 180,E1 6150.222,E2 6150.222} C_VEL
LIN {X 0,Y 490.66,Z 462.44,A -85,B 0,C 180,E1 6155.89,E2 6155.89} C_VEL
LIN {X 0,Y 490.506,Z 462.44,A -85,B 0,C 180,E1 6162.196,E2 6162.196} C_VEL
LIN {X 0,Y 490.506,Z 462.44,A -85,B 0,C 180,E1 6167.795,E2 6167.795} C_VEL
LIN {X 0,Y 490.659,Z 462.44,A -85,B 0,C 180,E1 6171.889,E2 6171.889} C_VEL
LIN {X 0,Y 493.165,Z 468.162,A -85,B 0,C 180,E1 6172.293,E2 6172.293} C_VEL
LIN {X 0,Y 507.11,Z 494.772,A -85,B 0,C 180,E1 6174.177,E2 6174.177} C_VEL
LIN {X 0,Y 510.28,Z 503.111,A -85,B 0,C 180,E1 6174.624,E2 6174.624} C_VEL
LIN {X 0,Y 508.743,Z 545.227,A -85,B 0,C 180,E1 6175.674,E2 6175.674} C_VEL
LIN {X 0,Y 506.056,Z 582.975,A -85,B 0,C 180,E1 6177.3,E2 6177.3} C_VEL
LIN {X 0,Y 503.107,Z 618.455,A -85,B 0,C 180,E1 6179.478,E2 6179.478} C_VEL
LIN {X 0,Y 499.763,Z 653.035,A -85,B 0,C 180,E1 6182.397,E2 6182.397} C_VEL
LIN {X 0,Y 496.814,Z 683.001,A -85,B 0,C 180,E1 6185.767,E2 6185.767} C_VEL
LIN {X 0,Y 494.392,Z 708.944,A -85,B 0,C 180,E1 6189.596,E2 6189.596} C_VEL
LIN {X 0,Y 492.899,Z 728.994,A -85,B 0,C 180,E1 6193.492,E2 6193.492} C_VEL
LIN {X 0,Y 492.021,Z 744.551,A -85,B 0,C 180,E1 6197.56,E2 6197.56} C_VEL
LIN {X 0,Y 491.681,Z 756.135,A -85,B 0,C 180,E1 6202.034,E2 6202.034} C_VEL
LIN {X 0,Y 491.491,Z 762.443,A -85,B 0,C 180,E1 6206.468,E2 6206.468} C_VEL
LIN {X 0,Y 491.533,Z 763.995,A -85,B 0,C 180,E1 6210,E2 6210} C_VEL
LIN {X 0,Y 491.518,Z 762.355,A -85,B 0,C 180,E1 6213.532,E2 6213.532} C_VEL
LIN {X 0,Y 491.731,Z 755.942,A -85,B 0,C 180,E1 6217.965,E2 6217.965} C_VEL
LIN {X 0,Y 492.147,Z 744.243,A -85,B 0,C 180,E1 6222.437,E2 6222.437} C_VEL
LIN {X 0,Y 493.131,Z 726.52,A -85,B 0,C 180,E1 6226.959,E2 6226.959} C_VEL
LIN {X 0,Y 494.835,Z 704.045,A -85,B 0,C 180,E1 6231.123,E2 6231.123} C_VEL
LIN {X 0,Y 497.322,Z 677.533,A -85,B 0,C 180,E1 6234.831,E2 6234.831} C_VEL
LIN {X 0,Y 500.42,Z 646.13,A -85,B 0,C 180,E1 6238.167,E2 6238.167} C_VEL
LIN {X 0,Y 503.582,Z 612.004,A -85,B 0,C 180,E1 6240.884,E2 6240.884} C_VEL
LIN {X 0,Y 506.708,Z 573.321,A -85,B 0,C 180,E1 6243.101,E2 6243.101} C_VEL
LIN {X 0,Y 509.293,Z 534.485,A -85,B 0,C 180,E1 6244.571,E2 6244.571} C_VEL
LIN {X 0,Y 509.861,Z 501.537,A -85,B 0,C 180,E1 6245.353,E2 6245.353} C_VEL
LIN {X 0,Y 496.121,Z 473.402,A -85,B 0,C 180,E1 6247.208,E2 6247.208} C_VEL
LIN {X 0,Y 490.691,Z 463.268,A -85,B 0,C 180,E1 6247.955,E2 6247.955} C_VEL
LIN {X 0,Y 490.608,Z 462.44,A -85,B 0,C 180,E1 6248.116,E2 6248.116} C_VEL
LIN {X 0,Y 490.568,Z 462.44,A -85,B 0,C 180,E1 6254.782,E2 6254.782} C_VEL
LIN {X 0,Y 490.546,Z 462.44,A -85,B 0,C 180,E1 6260.503,E2 6260.503} C_VEL
LIN {X 0,Y 490.589,Z 462.44,A -85,B 0,C 180,E1 6266.441,E2 6266.441} C_VEL
LIN {X 0,Y 490.712,Z 462.44,A -85,B 0,C 180,E1 6272.434,E2 6272.434} C_VEL
LIN {X 0,Y 490.896,Z 462.44,A -85,B 0,C 180,E1 6278.28,E2 6278.28} C_VEL
LIN {X 0,Y 491.067,Z 462.44,A -85,B 0,C 180,E1 6283.892,E2 6283.892} C_VEL
LIN {X 0,Y 491.171,Z 462.44,A -85,B 0,C 180,E1 6289.343,E2 6289.343} C_VEL
LIN {X 0,Y 491.249,Z 462.44,A -85,B 0,C 180,E1 6294.696,E2 6294.696} C_VEL
LIN {X 0,Y 491.402,Z 462.44,A -85,B 0,C 180,E1 6300.001,E2 6300.001} C_VEL
LIN {X 0,Y 491.293,Z 462.44,A -85,B 0,C 180,E1 6305.305,E2 6305.305} C_VEL
LIN {X 0,Y 491.152,Z 462.44,A -85,B 0,C 180,E1 6310.659,E2 6310.659} C_VEL
LIN {X 0,Y 490.952,Z 462.44,A -85,B 0,C 180,E1 6317.047,E2 6317.047} C_VEL
LIN {X 0,Y 490.869,Z 462.44,A -85,B 0,C 180,E1 6323.639,E2 6323.639} C_VEL
LIN {X 0,Y 490.631,Z 462.44,A -85,B 0,C 180,E1 6330.219,E2 6330.219} C_VEL
LIN {X 0,Y 490.577,Z 462.44,A -85,B 0,C 180,E1 6336.633,E2 6336.633} C_VEL
LIN {X 0,Y 490.687,Z 462.44,A -85,B 0,C 180,E1 6342.75,E2 6342.75} C_VEL
LIN {X 0,Y 490.63,Z 462.44,A -85,B 0,C 180,E1 6346.615,E2 6346.615} C_VEL
LIN {X 0,Y 491.208,Z 465.964,A -85,B 0,C 180,E1 6347.142,E2 6347.142} C_VEL
LIN {X 0,Y 493.314,Z 483.971,A -85,B 0,C 180,E1 6347.725,E2 6347.725} C_VEL
LIN {X 0,Y 508.397,Z 511.195,A -85,B 0,C 180,E1 6349.538,E2 6349.538} C_VEL
LIN {X 0,Y 506.355,Z 553.091,A -85,B 0,C 180,E1 6350.679,E2 6350.679} C_VEL
LIN {X 0,Y 503.386,Z 593.206,A -85,B 0,C 180,E1 6352.442,E2 6352.442} C_VEL
LIN {X 0,Y 499.51,Z 630.559,A -85,B 0,C 180,E1 6354.835,E2 6354.835} C_VEL
LIN {X 0,Y 495.137,Z 667.578,A -85,B 0,C 180,E1 6358.039,E2 6358.039} C_VEL
LIN {X 0,Y 491.049,Z 701.262,A -85,B 0,C 180,E1 6361.896,E2 6361.896} C_VEL
LIN {X 0,Y 487.834,Z 730.033,A -85,B 0,C 180,E1 6366.203,E2 6366.203} C_VEL
LIN {X 0,Y 485.528,Z 753.844,A -85,B 0,C 180,E1 6370.886,E2 6370.886} C_VEL
LIN {X 0,Y 484.392,Z 771.817,A -85,B 0,C 180,E1 6375.676,E2 6375.676} C_VEL
LIN {X 0,Y 483.859,Z 784.247,A -85,B 0,C 180,E1 6380.487,E2 6380.487} C_VEL
LIN {X 0,Y 483.757,Z 790.904,A -85,B 0,C 180,E1 6384.612,E2 6384.612} C_VEL
LIN {X 0,Y 483.725,Z 793.657,A -85,B 0,C 180,E1 6388.206,E2 6388.206} C_VEL
LIN {X 0,Y 483.612,Z 793.657,A -85,B 0,C 180,E1 6391.794,E2 6391.794} C_VEL
LIN {X 0,Y 483.744,Z 789.703,A -85,B 0,C 180,E1 6396.289,E2 6396.289} C_VEL
LIN {X 0,Y 483.967,Z 781.435,A -85,B 0,C 180,E1 6400.819,E2 6400.819} C_VEL
LIN {X 0,Y 484.669,Z 766.678,A -85,B 0,C 180,E1 6405.864,E2 6405.864} C_VEL
LIN {X 0,Y 486.257,Z 746.056,A -85,B 0,C 180,E1 6410.799,E2 6410.799} C_VEL
LIN {X 0,Y 488.922,Z 719.927,A -85,B 0,C 180,E1 6415.448,E2 6415.448} C_VEL
LIN {X 0,Y 492.568,Z 688.905,A -85,B 0,C 180,E1 6419.648,E2 6419.648} C_VEL
LIN {X 0,Y 496.998,Z 652.518,A -85,B 0,C 180,E1 6423.378,E2 6423.378} C_VEL
LIN {X 0,Y 501.348,Z 613.83,A -85,B 0,C 180,E1 6426.335,E2 6426.335} C_VEL
LIN {X 0,Y 504.848,Z 576.208,A -85,B 0,C 180,E1 6428.39,E2 6428.39} C_VEL
LIN {X 0,Y 507.464,Z 535.071,A -85,B 0,C 180,E1 6429.887,E2 6429.887} C_VEL
LIN {X 0,Y 508.14,Z 510.68,A -85,B 0,C 180,E1 6430.494,E2 6430.494} C_VEL
LIN {X 0,Y 482.821,Z 463.61,A -85,B 0,C 180,E1 6433.641,E2 6433.641} C_VEL
LIN {X 0,Y 482.698,Z 462.44,A -85,B 0,C 180,E1 6433.83,E2 6433.83} C_VEL
LIN {X 0,Y 482.692,Z 462.44,A -85,B 0,C 180,E1 6438.837,E2 6438.837} C_VEL
LIN {X 0,Y 482.635,Z 462.44,A -85,B 0,C 180,E1 6444.654,E2 6444.654} C_VEL
LIN {X 0,Y 482.729,Z 462.44,A -85,B 0,C 180,E1 6449.88,E2 6449.88} C_VEL
LIN {X 0,Y 482.897,Z 462.44,A -85,B 0,C 180,E1 6455.947,E2 6455.947} C_VEL
LIN {X 0,Y 483.061,Z 462.44,A -85,B 0,C 180,E1 6461.734,E2 6461.734} C_VEL
LIN {X 0,Y 482.978,Z 462.44,A -85,B 0,C 180,E1 6467.324,E2 6467.324} C_VEL
LIN {X 0,Y 483.335,Z 462.44,A -85,B 0,C 180,E1 6472.801,E2 6472.801} C_VEL
LIN {X 0,Y 483.611,Z 462.44,A -85,B 0,C 180,E1 6478.205,E2 6478.205} C_VEL
LIN {X 0,Y 483.449,Z 462.44,A -85,B 0,C 180,E1 6483.59,E2 6483.59} C_VEL
LIN {X 0,Y 483.255,Z 462.44,A -85,B 0,C 180,E1 6489.011,E2 6489.011} C_VEL
LIN {X 0,Y 483.108,Z 462.44,A -85,B 0,C 180,E1 6494.518,E2 6494.518} C_VEL
LIN {X 0,Y 482.98,Z 462.44,A -85,B 0,C 180,E1 6500.169,E2 6500.169} C_VEL
LIN {X 0,Y 482.822,Z 462.44,A -85,B 0,C 180,E1 6506.038,E2 6506.038} C_VEL
LIN {X 0,Y 482.801,Z 462.44,A -85,B 0,C 180,E1 6512.213,E2 6512.213} C_VEL
LIN {X 0,Y 482.688,Z 462.44,A -85,B 0,C 180,E1 6518.351,E2 6518.351} C_VEL
LIN {X 0,Y 482.484,Z 462.44,A -85,B 0,C 180,E1 6523.798,E2 6523.798} C_VEL
LIN {X 0,Y 482.713,Z 462.44,A -85,B 0,C 180,E1 6531.038,E2 6531.038} C_VEL
LIN {X 0,Y 485.188,Z 468.182,A -85,B 0,C 180,E1 6531.438,E2 6531.438} C_VEL
LIN {X 0,Y 500.478,Z 496.205,A -85,B 0,C 180,E1 6533.557,E2 6533.557} C_VEL
LIN {X 0,Y 504.178,Z 504.696,A -85,B 0,C 180,E1 6534.077,E2 6534.077} C_VEL
LIN {X 0,Y 502.452,Z 546.631,A -85,B 0,C 180,E1 6535.154,E2 6535.154} C_VEL
LIN {X 0,Y 499.545,Z 584.409,A -85,B 0,C 180,E1 6536.819,E2 6536.819} C_VEL
LIN {X 0,Y 496.013,Z 619.998,A -85,B 0,C 180,E1 6539.121,E2 6539.121} C_VEL
LIN {X 0,Y 492.634,Z 652.726,A -85,B 0,C 180,E1 6541.93,E2 6541.93} C_VEL
LIN {X 0,Y 489.465,Z 682.542,A -85,B 0,C 180,E1 6545.316,E2 6545.316} C_VEL
LIN {X 0,Y 486.827,Z 708.511,A -85,B 0,C 180,E1 6549.188,E2 6549.188} C_VEL
LIN {X 0,Y 485.19,Z 728.992,A -85,B 0,C 180,E1 6553.222,E2 6553.222} C_VEL
LIN {X 0,Y 484.121,Z 745.91,A -85,B 0,C 180,E1 6557.812,E2 6557.812} C_VEL
LIN {X 0,Y 483.804,Z 756.133,A -85,B 0,C 180,E1 6561.904,E2 6561.904} C_VEL
LIN {X 0,Y 483.593,Z 762.442,A -85,B 0,C 180,E1 6566.41,E2 6566.41} C_VEL
LIN {X 0,Y 483.65,Z 763.995,A -85,B 0,C 180,E1 6570,E2 6570} C_VEL
LIN {X 0,Y 483.618,Z 762.356,A -85,B 0,C 180,E1 6573.59,E2 6573.59} C_VEL
LIN {X 0,Y 483.857,Z 755.944,A -85,B 0,C 180,E1 6578.095,E2 6578.095} C_VEL
LIN {X 0,Y 484.309,Z 744.245,A -85,B 0,C 180,E1 6582.641,E2 6582.641} C_VEL
LIN {X 0,Y 485.356,Z 726.574,A -85,B 0,C 180,E1 6587.229,E2 6587.229} C_VEL
LIN {X 0,Y 487.298,Z 704.129,A -85,B 0,C 180,E1 6591.453,E2 6591.453} C_VEL
LIN {X 0,Y 490.006,Z 677.187,A -85,B 0,C 180,E1 6595.272,E2 6595.272} C_VEL
LIN {X 0,Y 493.289,Z 646.514,A -85,B 0,C 180,E1 6598.574,E2 6598.574} C_VEL
LIN {X 0,Y 496.909,Z 610.937,A -85,B 0,C 180,E1 6601.453,E2 6601.453} C_VEL
LIN {X 0,Y 500.253,Z 574.959,A -85,B 0,C 180,E1 6603.584,E2 6603.584} C_VEL
LIN {X 0,Y 503.069,Z 535.903,A -85,B 0,C 180,E1 6605.099,E2 6605.099} C_VEL
LIN {X 0,Y 503.842,Z 504.479,A -85,B 0,C 180,E1 6605.87,E2 6605.87} C_VEL
LIN {X 0,Y 491.049,Z 478.357,A -85,B 0,C 180,E1 6607.638,E2 6607.638} C_VEL
LIN {X 0,Y 482.838,Z 464.004,A -85,B 0,C 180,E1 6608.806,E2 6608.806} C_VEL
LIN {X 0,Y 482.666,Z 462.44,A -85,B 0,C 180,E1 6608.859,E2 6608.859} C_VEL
LIN {X 0,Y 482.588,Z 462.44,A -85,B 0,C 180,E1 6613.819,E2 6613.819} C_VEL
LIN {X 0,Y 482.617,Z 462.44,A -85,B 0,C 180,E1 6618.848,E2 6618.848} C_VEL
LIN {X 0,Y 482.6,Z 462.44,A -85,B 0,C 180,E1 6624.661,E2 6624.661} C_VEL
LIN {X 0,Y 482.717,Z 462.44,A -85,B 0,C 180,E1 6629.881,E2 6629.881} C_VEL
LIN {X 0,Y 482.88,Z 462.44,A -85,B 0,C 180,E1 6635.948,E2 6635.948} C_VEL
LIN {X 0,Y 483.063,Z 462.44,A -85,B 0,C 180,E1 6641.736,E2 6641.736} C_VEL
LIN {X 0,Y 483.194,Z 462.44,A -85,B 0,C 180,E1 6647.332,E2 6647.332} C_VEL
LIN {X 0,Y 483.261,Z 462.44,A -85,B 0,C 180,E1 6652.802,E2 6652.802} C_VEL
LIN {X 0,Y 483.416,Z 462.44,A -85,B 0,C 180,E1 6658.206,E2 6658.206} C_VEL
LIN {X 0,Y 483.37,Z 462.44,A -85,B 0,C 180,E1 6663.592,E2 6663.592} C_VEL
LIN {X 0,Y 483.213,Z 462.44,A -85,B 0,C 180,E1 6669.014,E2 6669.014} C_VEL
LIN {X 0,Y 483.113,Z 462.44,A -85,B 0,C 180,E1 6674.52,E2 6674.52} C_VEL
LIN {X 0,Y 482.98,Z 462.44,A -85,B 0,C 180,E1 6680.171,E2 6680.171} C_VEL
LIN {X 0,Y 482.887,Z 462.44,A -85,B 0,C 180,E1 6686.037,E2 6686.037} C_VEL
LIN {X 0,Y 482.725,Z 462.44,A -85,B 0,C 180,E1 6692.221,E2 6692.221} C_VEL
LIN {X 0,Y 482.682,Z 462.44,A -85,B 0,C 180,E1 6698.853,E2 6698.853} C_VEL
LIN {X 0,Y 482.685,Z 462.44,A -85,B 0,C 180,E1 6703.823,E2 6703.823} C_VEL
LIN {X 0,Y 482.72,Z 462.44,A -85,B 0,C 180,E1 6706.302,E2 6706.302} C_VEL
LIN {X 0,Y 489.723,Z 477.148,A -85,B 0,C 180,E1 6707.276,E2 6707.276} C_VEL
LIN {X 0,Y 493.314,Z 483.971,A -85,B 0,C 180,E1 6707.725,E2 6707.725} C_VEL
LIN {X 0,Y 500.309,Z 503.241,A -85,B 0,C 180,E1 6708.685,E2 6708.685} C_VEL
LIN {X 0,Y 501.878,Z 515.829,A -85,B 0,C 180,E1 6709.1,E2 6709.1} C_VEL
LIN {X 0,Y 499.359,Z 559.793,A -85,B 0,C 180,E1 6710.399,E2 6710.399} C_VEL
LIN {X 0,Y 495.633,Z 603.329,A -85,B 0,C 180,E1 6712.491,E2 6712.491} C_VEL
LIN {X 0,Y 491.644,Z 640.163,A -85,B 0,C 180,E1 6715.033,E2 6715.033} C_VEL
LIN {X 0,Y 486.865,Z 678.077,A -85,B 0,C 180,E1 6718.632,E2 6718.632} C_VEL
LIN {X 0,Y 482.594,Z 711.195,A -85,B 0,C 180,E1 6722.818,E2 6722.818} C_VEL
LIN {X 0,Y 479.483,Z 738.361,A -85,B 0,C 180,E1 6727.325,E2 6727.325} C_VEL
LIN {X 0,Y 477.417,Z 761.139,A -85,B 0,C 180,E1 6732.367,E2 6732.367} C_VEL
LIN {X 0,Y 476.305,Z 776.767,A -85,B 0,C 180,E1 6737.143,E2 6737.143} C_VEL
LIN {X 0,Y 475.868,Z 786.917,A -85,B 0,C 180,E1 6741.768,E2 6741.768} C_VEL
LIN {X 0,Y 475.737,Z 792.627,A -85,B 0,C 180,E1 6746.35,E2 6746.35} C_VEL
LIN {X 0,Y 475.767,Z 794,A -85,B 0,C 180,E1 6750,E2 6750} C_VEL
LIN {X 0,Y 475.7,Z 792.628,A -85,B 0,C 180,E1 6753.65,E2 6753.65} C_VEL
LIN {X 0,Y 475.884,Z 786.917,A -85,B 0,C 180,E1 6758.232,E2 6758.232} C_VEL
LIN {X 0,Y 476.225,Z 776.768,A -85,B 0,C 180,E1 6762.86,E2 6762.86} C_VEL
LIN {X 0,Y 477.431,Z 759.953,A -85,B 0,C 180,E1 6767.95,E2 6767.95} C_VEL
LIN {X 0,Y 479.56,Z 737.323,A -85,B 0,C 180,E1 6772.878,E2 6772.878} C_VEL
LIN {X 0,Y 482.909,Z 708.855,A -85,B 0,C 180,E1 6777.518,E2 6777.518} C_VEL
LIN {X 0,Y 487.195,Z 675.715,A -85,B 0,C 180,E1 6781.618,E2 6781.618} C_VEL
LIN {X 0,Y 491.809,Z 639.03,A -85,B 0,C 180,E1 6785.054,E2 6785.054} C_VEL
LIN {X 0,Y 495.97,Z 601.143,A -85,B 0,C 180,E1 6787.631,E2 6787.631} C_VEL
LIN {X 0,Y 499.598,Z 557.538,A -85,B 0,C 180,E1 6789.679,E2 6789.679} C_VEL
LIN {X 0,Y 501.489,Z 513.184,A -85,B 0,C 180,E1 6790.997,E2 6790.997} C_VEL
LIN {X 0,Y 474.924,Z 464.149,A -85,B 0,C 180,E1 6794.43,E2 6794.43} C_VEL
LIN {X 0,Y 474.708,Z 462.44,A -85,B 0,C 180,E1 6794.565,E2 6794.565} C_VEL
LIN {X 0,Y 474.697,Z 462.44,A -85,B 0,C 180,E1 6800.366,E2 6800.366} C_VEL
LIN {X 0,Y 474.706,Z 462.44,A -85,B 0,C 180,E1 6806.027,E2 6806.027} C_VEL
LIN {X 0,Y 474.815,Z 462.44,A -85,B 0,C 180,E1 6811.426,E2 6811.426} C_VEL
LIN {X 0,Y 475.04,Z 462.44,A -85,B 0,C 180,E1 6817.569,E2 6817.569} C_VEL
LIN {X 0,Y 475.091,Z 462.44,A -85,B 0,C 180,E1 6823.333,E2 6823.333} C_VEL
LIN {X 0,Y 475.176,Z 462.44,A -85,B 0,C 180,E1 6828.978,E2 6828.978} C_VEL
LIN {X 0,Y 475.475,Z 462.44,A -85,B 0,C 180,E1 6834.518,E2 6834.518} C_VEL
LIN {X 0,Y 475.568,Z 462.44,A -85,B 0,C 180,E1 6839.999,E2 6839.999} C_VEL
LIN {X 0,Y 475.417,Z 462.44,A -85,B 0,C 180,E1 6845.481,E2 6845.481} C_VEL
LIN {X 0,Y 475.255,Z 462.44,A -85,B 0,C 180,E1 6851.018,E2 6851.018} C_VEL
LIN {X 0,Y 475.086,Z 462.44,A -85,B 0,C 180,E1 6857.036,E2 6857.036} C_VEL
LIN {X 0,Y 474.985,Z 462.44,A -85,B 0,C 180,E1 6862.487,E2 6862.487} C_VEL
LIN {X 0,Y 474.79,Z 462.44,A -85,B 0,C 180,E1 6868.573,E2 6868.573} C_VEL
LIN {X 0,Y 474.823,Z 462.44,A -85,B 0,C 180,E1 6875.023,E2 6875.023} C_VEL
LIN {X 0,Y 474.625,Z 462.44,A -85,B 0,C 180,E1 6880.036,E2 6880.036} C_VEL
LIN {X 0,Y 474.499,Z 462.44,A -85,B 0,C 180,E1 6885.41,E2 6885.41} C_VEL
LIN {X 0,Y 474.809,Z 462.44,A -85,B 0,C 180,E1 6890.169,E2 6890.169} C_VEL
LIN {X 0,Y 477.391,Z 468.261,A -85,B 0,C 180,E1 6890.582,E2 6890.582} C_VEL
LIN {X 0,Y 494.952,Z 500.021,A -85,B 0,C 180,E1 6893.071,E2 6893.071} C_VEL
LIN {X 0,Y 498.111,Z 509.232,A -85,B 0,C 180,E1 6893.577,E2 6893.577} C_VEL
LIN {X 0,Y 496.109,Z 549.615,A -85,B 0,C 180,E1 6894.673,E2 6894.673} C_VEL
LIN {X 0,Y 493.005,Z 586.549,A -85,B 0,C 180,E1 6896.365,E2 6896.365} C_VEL
LIN {X 0,Y 489.236,Z 621.606,A -85,B 0,C 180,E1 6898.691,E2 6898.691} C_VEL
LIN {X 0,Y 485.233,Z 654.904,A -85,B 0,C 180,E1 6901.704,E2 6901.704} C_VEL
LIN {X 0,Y 481.814,Z 684.977,A -85,B 0,C 180,E1 6905.242,E2 6905.242} C_VEL
LIN {X 0,Y 479.05,Z 710.158,A -85,B 0,C 180,E1 6909.136,E2 6909.136} C_VEL
LIN {X 0,Y 477.291,Z 730.942,A -85,B 0,C 180,E1 6913.411,E2 6913.411} C_VEL
LIN {X 0,Y 476.264,Z 745.908,A -85,B 0,C 180,E1 6917.608,E2 6917.608} C_VEL
LIN {X 0,Y 475.931,Z 756.132,A -85,B 0,C 180,E1 6921.769,E2 6921.769} C_VEL
LIN {X 0,Y 475.69,Z 762.442,A -85,B 0,C 180,E1 6926.35,E2 6926.35} C_VEL
LIN {X 0,Y 475.749,Z 763.995,A -85,B 0,C 180,E1 6930,E2 6930} C_VEL
LIN {X 0,Y 475.714,Z 762.357,A -85,B 0,C 180,E1 6933.65,E2 6933.65} C_VEL
LIN {X 0,Y 475.985,Z 755.946,A -85,B 0,C 180,E1 6938.23,E2 6938.23} C_VEL
LIN {X 0,Y 476.479,Z 744.246,A -85,B 0,C 180,E1 6942.853,E2 6942.853} C_VEL
LIN {X 0,Y 477.584,Z 727.343,A -85,B 0,C 180,E1 6947.35,E2 6947.35} C_VEL
LIN {X 0,Y 479.747,Z 704.13,A -85,B 0,C 180,E1 6951.808,E2 6951.808} C_VEL
LIN {X 0,Y 482.773,Z 676.288,A -85,B 0,C 180,E1 6955.796,E2 6955.796} C_VEL
LIN {X 0,Y 486.6,Z 643.266,A -85,B 0,C 180,E1 6959.357,E2 6959.357} C_VEL
LIN {X 0,Y 490.687,Z 608.826,A -85,B 0,C 180,E1 6962.16,E2 6962.16} C_VEL
LIN {X 0,Y 494.464,Z 570.441,A -85,B 0,C 180,E1 6964.38,E2 6964.38} C_VEL
LIN {X 0,Y 497.321,Z 530.344,A -85,B 0,C 180,E1 6965.855,E2 6965.855} C_VEL
LIN {X 0,Y 497.774,Z 507.154,A -85,B 0,C 180,E1 6966.411,E2 6966.411} C_VEL
LIN {X 0,Y 485.55,Z 482.42,A -85,B 0,C 180,E1 6968.158,E2 6968.158} C_VEL
LIN {X 0,Y 474.725,Z 463.467,A -85,B 0,C 180,E1 6969.713,E2 6969.713} C_VEL
LIN {X 0,Y 474.658,Z 462.44,A -85,B 0,C 180,E1 6969.939,E2 6969.939} C_VEL
LIN {X 0,Y 474.613,Z 462.44,A -85,B 0,C 180,E1 6975.432,E2 6975.432} C_VEL
LIN {X 0,Y 474.632,Z 462.44,A -85,B 0,C 180,E1 6980.362,E2 6980.362} C_VEL
LIN {X 0,Y 474.68,Z 462.44,A -85,B 0,C 180,E1 6986.032,E2 6986.032} C_VEL
LIN {X 0,Y 474.804,Z 462.44,A -85,B 0,C 180,E1 6991.428,E2 6991.428} C_VEL
LIN {X 0,Y 475.033,Z 462.44,A -85,B 0,C 180,E1 6997.571,E2 6997.571} C_VEL
LIN {X 0,Y 475.195,Z 462.44,A -85,B 0,C 180,E1 7003.338,E2 7003.338} C_VEL
LIN {X 0,Y 475.316,Z 462.44,A -85,B 0,C 180,E1 7008.984,E2 7008.984} C_VEL
LIN {X 0,Y 475.432,Z 462.44,A -85,B 0,C 180,E1 7014.519,E2 7014.519} C_VEL
LIN {X 0,Y 475.631,Z 462.44,A -85,B 0,C 180,E1 7020.001,E2 7020.001} C_VEL
LIN {X 0,Y 475.478,Z 462.44,A -85,B 0,C 180,E1 7025.482,E2 7025.482} C_VEL
LIN {X 0,Y 475.291,Z 462.44,A -85,B 0,C 180,E1 7031.019,E2 7031.019} C_VEL
LIN {X 0,Y 475.082,Z 462.44,A -85,B 0,C 180,E1 7037.034,E2 7037.034} C_VEL
LIN {X 0,Y 475.036,Z 462.44,A -85,B 0,C 180,E1 7042.486,E2 7042.486} C_VEL
LIN {X 0,Y 474.819,Z 462.44,A -85,B 0,C 180,E1 7048.574,E2 7048.574} C_VEL
LIN {X 0,Y 474.724,Z 462.44,A -85,B 0,C 180,E1 7055.034,E2 7055.034} C_VEL
LIN {X 0,Y 474.69,Z 462.44,A -85,B 0,C 180,E1 7060.045,E2 7060.045} C_VEL
LIN {X 0,Y 474.718,Z 462.528,A -85,B 0,C 180,E1 7065.515,E2 7065.515} C_VEL
LIN {X 0,Y 479.139,Z 472.069,A -85,B 0,C 180,E1 7066.166,E2 7066.166} C_VEL
LIN {X 0,Y 501.862,Z 513.956,A -85,B 0,C 180,E1 7069.051,E2 7069.051} C_VEL
LIN {X 0,Y 501.878,Z 515.829,A -85,B 0,C 180,E1 7069.1,E2 7069.1} C_VEL
LIN {X 0,Y 499.54,Z 528.644,A -85,B 0,C 180,E1 7069.253,E2 7069.253} C_VEL
LIN {X 0,Y 493.873,Z 547.638,A -85,B 0,C 180,E1 7069.445,E2 7069.445} C_VEL
LIN {X 0,Y 493.614,Z 549.688,A -85,B 0,C 180,E1 7069.509,E2 7069.509} C_VEL
LIN {X 0,Y 490.278,Z 590.983,A -85,B 0,C 180,E1 7071.311,E2 7071.311} C_VEL
LIN {X 0,Y 486.201,Z 629.558,A -85,B 0,C 180,E1 7073.722,E2 7073.722} C_VEL
LIN {X 0,Y 481.835,Z 664.119,A -85,B 0,C 180,E1 7076.661,E2 7076.661} C_VEL
LIN {X 0,Y 476.958,Z 698.765,A -85,B 0,C 180,E1 7080.628,E2 7080.628} C_VEL
LIN {X 0,Y 473.043,Z 728.686,A -85,B 0,C 180,E1 7085.158,E2 7085.158} C_VEL
LIN {X 0,Y 470.208,Z 752.835,A -85,B 0,C 180,E1 7089.993,E2 7089.993} C_VEL
LIN {X 0,Y 468.809,Z 769.76,A -85,B 0,C 180,E1 7094.547,E2 7094.547} C_VEL
LIN {X 0,Y 468.131,Z 781.434,A -85,B 0,C 180,E1 7098.81,E2 7098.81} C_VEL
LIN {X 0,Y 467.914,Z 789.702,A -85,B 0,C 180,E1 7103.497,E2 7103.497} C_VEL
LIN {X 0,Y 467.925,Z 793.657,A -85,B 0,C 180,E1 7108.146,E2 7108.146} C_VEL
LIN {X 0,Y 467.805,Z 793.657,A -85,B 0,C 180,E1 7111.855,E2 7111.855} C_VEL
LIN {X 0,Y 467.936,Z 789.703,A -85,B 0,C 180,E1 7116.503,E2 7116.503} C_VEL
LIN {X 0,Y 468.204,Z 781.434,A -85,B 0,C 180,E1 7121.188,E2 7121.188} C_VEL
LIN {X 0,Y 469.099,Z 766.68,A -85,B 0,C 180,E1 7126.405,E2 7126.405} C_VEL
LIN {X 0,Y 471.099,Z 745.561,A -85,B 0,C 180,E1 7131.611,E2 7131.611} C_VEL
LIN {X 0,Y 474.102,Z 719.93,A -85,B 0,C 180,E1 7136.303,E2 7136.303} C_VEL
LIN {X 0,Y 478.511,Z 688.188,A -85,B 0,C 180,E1 7140.702,E2 7140.702} C_VEL
LIN {X 0,Y 483.401,Z 652.712,A -85,B 0,C 180,E1 7144.422,E2 7144.422} C_VEL
LIN {X 0,Y 487.917,Z 614.585,A -85,B 0,C 180,E1 7147.31,E2 7147.31} C_VEL
LIN {X 0,Y 491.908,Z 573.904,A -85,B 0,C 180,E1 7149.524,E2 7149.524} C_VEL
LIN {X 0,Y 494.723,Z 533.476,A -85,B 0,C 180,E1 7150.994,E2 7150.994} C_VEL
LIN {X 0,Y 495.193,Z 516.414,A -85,B 0,C 180,E1 7151.456,E2 7151.456} C_VEL
LIN {X 0,Y 466.871,Z 463.387,A -85,B 0,C 180,E1 7155.325,E2 7155.325} C_VEL
LIN {X 0,Y 466.793,Z 462.44,A -85,B 0,C 180,E1 7155.53,E2 7155.53} C_VEL
LIN {X 0,Y 466.743,Z 462.44,A -85,B 0,C 180,E1 7161.953,E2 7161.953} C_VEL
LIN {X 0,Y 466.796,Z 462.44,A -85,B 0,C 180,E1 7168.739,E2 7168.739} C_VEL
LIN {X 0,Y 467.052,Z 462.44,A -85,B 0,C 180,E1 7175.194,E2 7175.194} C_VEL
LIN {X 0,Y 467.187,Z 462.44,A -85,B 0,C 180,E1 7181.09,E2 7181.09} C_VEL
LIN {X 0,Y 467.129,Z 462.44,A -85,B 0,C 180,E1 7186.886,E2 7186.886} C_VEL
LIN {X 0,Y 467.483,Z 462.44,A -85,B 0,C 180,E1 7192.556,E2 7192.556} C_VEL
LIN {X 0,Y 467.799,Z 462.44,A -85,B 0,C 180,E1 7198.144,E2 7198.144} C_VEL
LIN {X 0,Y 467.623,Z 462.44,A -85,B 0,C 180,E1 7203.712,E2 7203.712} C_VEL
LIN {X 0,Y 467.425,Z 462.44,A -85,B 0,C 180,E1 7209.319,E2 7209.319} C_VEL
LIN {X 0,Y 467.233,Z 462.44,A -85,B 0,C 180,E1 7215.023,E2 7215.023} C_VEL
LIN {X 0,Y 467.1,Z 462.44,A -85,B 0,C 180,E1 7220.886,E2 7220.886} C_VEL
LIN {X 0,Y 466.89,Z 462.44,A -85,B 0,C 180,E1 7226.997,E2 7226.997} C_VEL
LIN {X 0,Y 466.88,Z 462.44,A -85,B 0,C 180,E1 7233.452,E2 7233.452} C_VEL
LIN {X 0,Y 466.673,Z 462.44,A -85,B 0,C 180,E1 7240.452,E2 7240.452} C_VEL
LIN {X 0,Y 466.617,Z 462.44,A -85,B 0,C 180,E1 7247.044,E2 7247.044} C_VEL
LIN {X 0,Y 466.768,Z 462.44,A -85,B 0,C 180,E1 7249.248,E2 7249.248} C_VEL
LIN {X 0,Y 469.143,Z 468.026,A -85,B 0,C 180,E1 7249.651,E2 7249.651} C_VEL
LIN {X 0,Y 489.289,Z 503.474,A -85,B 0,C 180,E1 7252.545,E2 7252.545} C_VEL
LIN {X 0,Y 492.101,Z 511.415,A -85,B 0,C 180,E1 7253.015,E2 7253.015} C_VEL
LIN {X 0,Y 489.942,Z 551.352,A -85,B 0,C 180,E1 7254.136,E2 7254.136} C_VEL
LIN {X 0,Y 486.586,Z 588.164,A -85,B 0,C 180,E1 7255.861,E2 7255.861} C_VEL
LIN {X 0,Y 482.659,Z 621.917,A -85,B 0,C 180,E1 7258.145,E2 7258.145} C_VEL
LIN {X 0,Y 478.361,Z 654.659,A -85,B 0,C 180,E1 7261.15,E2 7261.15} C_VEL
LIN {X 0,Y 474.079,Z 687.798,A -85,B 0,C 180,E1 7265.216,E2 7265.216} C_VEL
LIN {X 0,Y 471.07,Z 714.299,A -85,B 0,C 180,E1 7269.54,E2 7269.54} C_VEL
LIN {X 0,Y 469.21,Z 734.754,A -85,B 0,C 180,E1 7274.08,E2 7274.08} C_VEL
LIN {X 0,Y 468.274,Z 749.821,A -85,B 0,C 180,E1 7278.813,E2 7278.813} C_VEL
LIN {X 0,Y 467.967,Z 759.285,A -85,B 0,C 180,E1 7283.498,E2 7283.498} C_VEL
LIN {X 0,Y 467.789,Z 763.61,A -85,B 0,C 180,E1 7288.145,E2 7288.145} C_VEL
LIN {X 0,Y 467.908,Z 763.559,A -85,B 0,C 180,E1 7291.854,E2 7291.854} C_VEL
LIN {X 0,Y 467.957,Z 759.158,A -85,B 0,C 180,E1 7296.503,E2 7296.503} C_VEL
LIN {X 0,Y 468.283,Z 749.602,A -85,B 0,C 180,E1 7301.187,E2 7301.187} C_VEL
LIN {X 0,Y 469.285,Z 734.428,A -85,B 0,C 180,E1 7305.917,E2 7305.917} C_VEL
LIN {X 0,Y 471.286,Z 712.514,A -85,B 0,C 180,E1 7310.696,E2 7310.696} C_VEL
LIN {X 0,Y 474.176,Z 687.165,A -85,B 0,C 180,E1 7314.778,E2 7314.778} C_VEL
LIN {X 0,Y 478.234,Z 655.244,A -85,B 0,C 180,E1 7318.702,E2 7318.702} C_VEL
LIN {X 0,Y 482.462,Z 622.666,A -85,B 0,C 180,E1 7321.714,E2 7321.714} C_VEL
LIN {X 0,Y 486.714,Z 586.713,A -85,B 0,C 180,E1 7324.133,E2 7324.133} C_VEL
LIN {X 0,Y 490.102,Z 550.258,A -85,B 0,C 180,E1 7325.805,E2 7325.805} C_VEL
LIN {X 0,Y 492.155,Z 514.225,A -85,B 0,C 180,E1 7326.827,E2 7326.827} C_VEL
LIN {X 0,Y 491.025,Z 508.048,A -85,B 0,C 180,E1 7327.082,E2 7327.082} C_VEL
LIN {X 0,Y 478.153,Z 483.084,A -85,B 0,C 180,E1 7328.962,E2 7328.962} C_VEL
LIN {X 0,Y 466.785,Z 463.729,A -85,B 0,C 180,E1 7330.612,E2 7330.612} C_VEL
LIN {X 0,Y 466.678,Z 462.44,A -85,B 0,C 180,E1 7330.83,E2 7330.83} C_VEL
LIN {X 0,Y 466.729,Z 462.44,A -85,B 0,C 180,E1 7337.065,E2 7337.065} C_VEL
LIN {X 0,Y 466.695,Z 462.44,A -85,B 0,C 180,E1 7341.951,E2 7341.951} C_VEL
LIN {X 0,Y 466.779,Z 462.44,A -85,B 0,C 180,E1 7348.74,E2 7348.74} C_VEL
LIN {X 0,Y 467.023,Z 462.44,A -85,B 0,C 180,E1 7355.201,E2 7355.201} C_VEL
LIN {X 0,Y 467.184,Z 462.44,A -85,B 0,C 180,E1 7361.093,E2 7361.093} C_VEL
LIN {X 0,Y 467.36,Z 462.44,A -85,B 0,C 180,E1 7366.895,E2 7366.895} C_VEL
LIN {X 0,Y 467.439,Z 462.44,A -85,B 0,C 180,E1 7372.557,E2 7372.557} C_VEL
LIN {X 0,Y 467.644,Z 462.44,A -85,B 0,C 180,E1 7378.146,E2 7378.146} C_VEL
LIN {X 0,Y 467.557,Z 462.44,A -85,B 0,C 180,E1 7383.714,E2 7383.714} C_VEL
LIN {X 0,Y 467.377,Z 462.44,A -85,B 0,C 180,E1 7389.322,E2 7389.322} C_VEL
LIN {X 0,Y 467.24,Z 462.44,A -85,B 0,C 180,E1 7395.025,E2 7395.025} C_VEL
LIN {X 0,Y 467.114,Z 462.44,A -85,B 0,C 180,E1 7400.888,E2 7400.888} C_VEL
LIN {X 0,Y 466.962,Z 462.44,A -85,B 0,C 180,E1 7406.995,E2 7406.995} C_VEL
LIN {X 0,Y 466.796,Z 462.44,A -85,B 0,C 180,E1 7413.461,E2 7413.461} C_VEL
LIN {X 0,Y 466.756,Z 462.44,A -85,B 0,C 180,E1 7420.446,E2 7420.446} C_VEL
LIN {X 0,Y 466.804,Z 462.44,A -85,B 0,C 180,E1 7424.614,E2 7424.614} C_VEL
LIN {X 0,Y 471.322,Z 472.2,A -85,B 0,C 180,E1 7425.353,E2 7425.353} C_VEL
LIN {X 0,Y 495.471,Z 516.866,A -85,B 0,C 180,E1 7428.581,E2 7428.581} C_VEL
LIN {X 0,Y 493.614,Z 549.688,A -85,B 0,C 180,E1 7429.509,E2 7429.509} C_VEL
LIN {X 0,Y 489.358,Z 560.792,A -85,B 0,C 180,E1 7429.627,E2 7429.627} C_VEL
LIN {X 0,Y 485.601,Z 570.373,A -85,B 0,C 180,E1 7429.781,E2 7429.781} C_VEL
LIN {X 0,Y 485.459,Z 571.763,A -85,B 0,C 180,E1 7429.837,E2 7429.837} C_VEL
LIN {X 0,Y 481.105,Z 613.99,A -85,B 0,C 180,E1 7432.131,E2 7432.131} C_VEL
LIN {X 0,Y 476.158,Z 654.169,A -85,B 0,C 180,E1 7435.229,E2 7435.229} C_VEL
LIN {X 0,Y 471.617,Z 686.781,A -85,B 0,C 180,E1 7438.619,E2 7438.619} C_VEL
LIN {X 0,Y 466.995,Z 718.362,A -85,B 0,C 180,E1 7443.004,E2 7443.004} C_VEL
LIN {X 0,Y 463.591,Z 745.178,A -85,B 0,C 180,E1 7447.938,E2 7447.938} C_VEL
LIN {X 0,Y 461.371,Z 766.682,A -85,B 0,C 180,E1 7453.312,E2 7453.312} C_VEL
LIN {X 0,Y 460.266,Z 781.433,A -85,B 0,C 180,E1 7458.616,E2 7458.616} C_VEL
LIN {X 0,Y 460.014,Z 789.702,A -85,B 0,C 180,E1 7463.385,E2 7463.385} C_VEL
LIN {X 0,Y 460.019,Z 793.657,A -85,B 0,C 180,E1 7468.114,E2 7468.114} C_VEL
LIN {X 0,Y 459.901,Z 793.657,A -85,B 0,C 180,E1 7471.887,E2 7471.887} C_VEL
LIN {X 0,Y 460.037,Z 789.703,A -85,B 0,C 180,E1 7476.615,E2 7476.615} C_VEL
LIN {X 0,Y 460.319,Z 781.434,A -85,B 0,C 180,E1 7481.383,E2 7481.383} C_VEL
LIN {X 0,Y 461.325,Z 766.681,A -85,B 0,C 180,E1 7486.69,E2 7486.69} C_VEL
LIN {X 0,Y 463.519,Z 745.175,A -85,B 0,C 180,E1 7492.065,E2 7492.065} C_VEL
LIN {X 0,Y 466.998,Z 718.363,A -85,B 0,C 180,E1 7496.995,E2 7496.995} C_VEL
LIN {X 0,Y 471.61,Z 686.754,A -85,B 0,C 180,E1 7501.385,E2 7501.385} C_VEL
LIN {X 0,Y 476.22,Z 654.149,A -85,B 0,C 180,E1 7504.769,E2 7504.769} C_VEL
LIN {X 0,Y 481.069,Z 615.266,A -85,B 0,C 180,E1 7507.775,E2 7507.775} C_VEL
LIN {X 0,Y 485.376,Z 573.794,A -85,B 0,C 180,E1 7510.064,E2 7510.064} C_VEL
LIN {X 0,Y 488.35,Z 533.324,A -85,B 0,C 180,E1 7511.543,E2 7511.543} C_VEL
LIN {X 0,Y 488.593,Z 519.119,A -85,B 0,C 180,E1 7511.954,E2 7511.954} C_VEL
LIN {X 0,Y 460.973,Z 467.802,A -85,B 0,C 180,E1 7515.904,E2 7515.904} C_VEL
LIN {X 0,Y 458.87,Z 462.44,A -85,B 0,C 180,E1 7516.377,E2 7516.377} C_VEL
LIN {X 0,Y 458.812,Z 462.44,A -85,B 0,C 180,E1 7522.376,E2 7522.376} C_VEL
LIN {X 0,Y 458.877,Z 462.44,A -85,B 0,C 180,E1 7529.083,E2 7529.083} C_VEL
LIN {X 0,Y 459.074,Z 462.44,A -85,B 0,C 180,E1 7534.613,E2 7534.613} C_VEL
LIN {X 0,Y 459.278,Z 462.44,A -85,B 0,C 180,E1 7540.752,E2 7540.752} C_VEL
LIN {X 0,Y 459.218,Z 462.44,A -85,B 0,C 180,E1 7546.656,E2 7546.656} C_VEL
LIN {X 0,Y 459.554,Z 462.44,A -85,B 0,C 180,E1 7552.427,E2 7552.427} C_VEL
LIN {X 0,Y 459.887,Z 462.44,A -85,B 0,C 180,E1 7558.112,E2 7558.112} C_VEL
LIN {X 0,Y 459.709,Z 462.44,A -85,B 0,C 180,E1 7563.775,E2 7563.775} C_VEL
LIN {X 0,Y 459.523,Z 462.44,A -85,B 0,C 180,E1 7569.481,E2 7569.481} C_VEL
LIN {X 0,Y 459.295,Z 462.44,A -85,B 0,C 180,E1 7575.289,E2 7575.289} C_VEL
LIN {X 0,Y 459.143,Z 462.44,A -85,B 0,C 180,E1 7581.265,E2 7581.265} C_VEL
LIN {X 0,Y 458.958,Z 462.44,A -85,B 0,C 180,E1 7587.503,E2 7587.503} C_VEL
LIN {X 0,Y 458.892,Z 462.44,A -85,B 0,C 180,E1 7594.114,E2 7594.114} C_VEL
LIN {X 0,Y 458.754,Z 462.44,A -85,B 0,C 180,E1 7600.613,E2 7600.613} C_VEL
LIN {X 0,Y 458.681,Z 462.44,A -85,B 0,C 180,E1 7606.563,E2 7606.563} C_VEL
LIN {X 0,Y 458.77,Z 462.44,A -85,B 0,C 180,E1 7608.304,E2 7608.304} C_VEL
LIN {X 0,Y 461.294,Z 468.195,A -85,B 0,C 180,E1 7608.735,E2 7608.735} C_VEL
LIN {X 0,Y 483.479,Z 506.559,A -85,B 0,C 180,E1 7611.984,E2 7611.984} C_VEL
LIN {X 0,Y 486.174,Z 512.809,A -85,B 0,C 180,E1 7612.417,E2 7612.417} C_VEL
LIN {X 0,Y 483.837,Z 553.044,A -85,B 0,C 180,E1 7613.579,E2 7613.579} C_VEL
LIN {X 0,Y 480.13,Z 590.919,A -85,B 0,C 180,E1 7615.414,E2 7615.414} C_VEL
LIN {X 0,Y 475.849,Z 624.626,A -85,B 0,C 180,E1 7617.769,E2 7617.769} C_VEL
LIN {X 0,Y 471.212,Z 656.973,A -85,B 0,C 180,E1 7620.842,E2 7620.842} C_VEL
LIN {X 0,Y 467,Z 686.384,A -85,B 0,C 180,E1 7624.558,E2 7624.558} C_VEL
LIN {X 0,Y 463.451,Z 714.297,A -85,B 0,C 180,E1 7629.188,E2 7629.188} C_VEL
LIN {X 0,Y 461.452,Z 734.752,A -85,B 0,C 180,E1 7633.805,E2 7633.805} C_VEL
LIN {X 0,Y 460.428,Z 749.819,A -85,B 0,C 180,E1 7638.62,E2 7638.62} C_VEL
LIN {X 0,Y 460.066,Z 759.284,A -85,B 0,C 180,E1 7643.385,E2 7643.385} C_VEL
LIN {X 0,Y 459.885,Z 763.61,A -85,B 0,C 180,E1 7648.113,E2 7648.113} C_VEL
LIN {X 0,Y 460.002,Z 763.559,A -85,B 0,C 180,E1 7651.886,E2 7651.886} C_VEL
LIN {X 0,Y 460.059,Z 759.159,A -85,B 0,C 180,E1 7656.615,E2 7656.615} C_VEL
LIN {X 0,Y 460.454,Z 749.604,A -85,B 0,C 180,E1 7661.379,E2 7661.379} C_VEL
LIN {X 0,Y 461.529,Z 734.432,A -85,B 0,C 180,E1 7666.192,E2 7666.192} C_VEL
LIN {X 0,Y 463.669,Z 712.517,A -85,B 0,C 180,E1 7671.052,E2 7671.052} C_VEL
LIN {X 0,Y 467.303,Z 684.099,A -85,B 0,C 180,E1 7675.682,E2 7675.682} C_VEL
LIN {X 0,Y 471.555,Z 654.596,A -85,B 0,C 180,E1 7679.326,E2 7679.326} C_VEL
LIN {X 0,Y 476.289,Z 620.746,A -85,B 0,C 180,E1 7682.463,E2 7682.463} C_VEL
LIN {X 0,Y 480.969,Z 582.623,A -85,B 0,C 180,E1 7684.981,E2 7684.981} C_VEL
LIN {X 0,Y 484.669,Z 542.409,A -85,B 0,C 180,E1 7686.711,E2 7686.711} C_VEL
LIN {X 0,Y 485.822,Z 512.565,A -85,B 0,C 180,E1 7687.534,E2 7687.534} C_VEL
LIN {X 0,Y 473.603,Z 488.64,A -85,B 0,C 180,E1 7689.36,E2 7689.36} C_VEL
LIN {X 0,Y 459.014,Z 464.209,A -85,B 0,C 180,E1 7691.526,E2 7691.526} C_VEL
LIN {X 0,Y 458.805,Z 462.44,A -85,B 0,C 180,E1 7691.622,E2 7691.622} C_VEL
LIN {X 0,Y 458.802,Z 462.44,A -85,B 0,C 180,E1 7696.556,E2 7696.556} C_VEL
LIN {X 0,Y 458.765,Z 462.44,A -85,B 0,C 180,E1 7702.383,E2 7702.383} C_VEL
LIN {X 0,Y 458.862,Z 462.44,A -85,B 0,C 180,E1 7709.086,E2 7709.086} C_VEL
LIN {X 0,Y 459.046,Z 462.44,A -85,B 0,C 180,E1 7714.613,E2 7714.613} C_VEL
LIN {X 0,Y 459.276,Z 462.44,A -85,B 0,C 180,E1 7720.754,E2 7720.754} C_VEL
LIN {X 0,Y 459.462,Z 462.44,A -85,B 0,C 180,E1 7726.666,E2 7726.666} C_VEL
LIN {X 0,Y 459.526,Z 462.44,A -85,B 0,C 180,E1 7732.428,E2 7732.428} C_VEL
LIN {X 0,Y 459.742,Z 462.44,A -85,B 0,C 180,E1 7738.114,E2 7738.114} C_VEL
LIN {X 0,Y 459.649,Z 462.44,A -85,B 0,C 180,E1 7743.778,E2 7743.778} C_VEL
LIN {X 0,Y 459.456,Z 462.44,A -85,B 0,C 180,E1 7749.484,E2 7749.484} C_VEL
LIN {X 0,Y 459.302,Z 462.44,A -85,B 0,C 180,E1 7755.291,E2 7755.291} C_VEL
LIN {X 0,Y 459.164,Z 462.44,A -85,B 0,C 180,E1 7761.267,E2 7761.267} C_VEL
LIN {X 0,Y 459.009,Z 462.44,A -85,B 0,C 180,E1 7767.502,E2 7767.502} C_VEL
LIN {X 0,Y 458.813,Z 462.44,A -85,B 0,C 180,E1 7774.408,E2 7774.408} C_VEL
LIN {X 0,Y 458.876,Z 462.44,A -85,B 0,C 180,E1 7781.29,E2 7781.29} C_VEL
LIN {X 0,Y 458.872,Z 462.838,A -85,B 0,C 180,E1 7783.74,E2 7783.74} C_VEL
LIN {X 0,Y 461.535,Z 468.356,A -85,B 0,C 180,E1 7784.175,E2 7784.175} C_VEL
LIN {X 0,Y 488.926,Z 520.965,A -85,B 0,C 180,E1 7788.129,E2 7788.129} C_VEL
LIN {X 0,Y 486.093,Z 562.851,A -85,B 0,C 180,E1 7789.457,E2 7789.457} C_VEL
LIN {X 0,Y 485.459,Z 571.763,A -85,B 0,C 180,E1 7789.837,E2 7789.837} C_VEL
LIN {X 0,Y 483.904,Z 579.99,A -85,B 0,C 180,E1 7790.136,E2 7790.136} C_VEL
LIN {X 0,Y 475.895,Z 602.055,A -85,B 0,C 180,E1 7790.875,E2 7790.875} C_VEL
LIN {X 0,Y 475.541,Z 604.001,A -85,B 0,C 180,E1 7790.986,E2 7790.986} C_VEL
LIN {X 0,Y 470.625,Z 643.262,A -85,B 0,C 180,E1 7793.794,E2 7793.794} C_VEL
LIN {X 0,Y 465.632,Z 679.281,A -85,B 0,C 180,E1 7797.284,E2 7797.284} C_VEL
LIN {X 0,Y 461.148,Z 708.652,A -85,B 0,C 180,E1 7801.033,E2 7801.033} C_VEL
LIN {X 0,Y 457.001,Z 736.616,A -85,B 0,C 180,E1 7805.784,E2 7805.784} C_VEL
LIN {X 0,Y 454.263,Z 758.798,A -85,B 0,C 180,E1 7810.801,E2 7810.801} C_VEL
LIN {X 0,Y 452.916,Z 774.926,A -85,B 0,C 180,E1 7815.788,E2 7815.788} C_VEL
LIN {X 0,Y 452.278,Z 785.329,A -85,B 0,C 180,E1 7820.364,E2 7820.364} C_VEL
LIN {X 0,Y 452.135,Z 790.904,A -85,B 0,C 180,E1 7824.234,E2 7824.234} C_VEL
LIN {X 0,Y 452.144,Z 793.657,A -85,B 0,C 180,E1 7828.081,E2 7828.081} C_VEL
LIN {X 0,Y 452.007,Z 793.657,A -85,B 0,C 180,E1 7831.92,E2 7831.92} C_VEL
LIN {X 0,Y 452.144,Z 789.703,A -85,B 0,C 180,E1 7836.731,E2 7836.731} C_VEL
LIN {X 0,Y 452.442,Z 781.434,A -85,B 0,C 180,E1 7841.583,E2 7841.583} C_VEL
LIN {X 0,Y 453.56,Z 766.682,A -85,B 0,C 180,E1 7846.984,E2 7846.984} C_VEL
LIN {X 0,Y 455.934,Z 745.173,A -85,B 0,C 180,E1 7852.452,E2 7852.452} C_VEL
LIN {X 0,Y 459.692,Z 718.362,A -85,B 0,C 180,E1 7857.46,E2 7857.46} C_VEL
LIN {X 0,Y 464.163,Z 689.026,A -85,B 0,C 180,E1 7861.597,E2 7861.597} C_VEL
LIN {X 0,Y 469.405,Z 653.107,A -85,B 0,C 180,E1 7865.349,E2 7865.349} C_VEL
LIN {X 0,Y 474.557,Z 613.526,A -85,B 0,C 180,E1 7868.413,E2 7868.413} C_VEL
LIN {X 0,Y 479.009,Z 571.83,A -85,B 0,C 180,E1 7870.695,E2 7870.695} C_VEL
LIN {X 0,Y 482.117,Z 532.078,A -85,B 0,C 180,E1 7872.137,E2 7872.137} C_VEL
LIN {X 0,Y 482.208,Z 522.2,A -85,B 0,C 180,E1 7872.438,E2 7872.438} C_VEL
LIN {X 0,Y 456.412,Z 473.414,A -85,B 0,C 180,E1 7876.319,E2 7876.319} C_VEL
LIN {X 0,Y 451.06,Z 463.944,A -85,B 0,C 180,E1 7877.191,E2 7877.191} C_VEL
LIN {X 0,Y 450.912,Z 462.44,A -85,B 0,C 180,E1 7877.304,E2 7877.304} C_VEL
LIN {X 0,Y 450.895,Z 462.44,A -85,B 0,C 180,E1 7883.701,E2 7883.701} C_VEL
LIN {X 0,Y 450.954,Z 462.44,A -85,B 0,C 180,E1 7889.761,E2 7889.761} C_VEL
LIN {X 0,Y 451.175,Z 462.44,A -85,B 0,C 180,E1 7896.254,E2 7896.254} C_VEL
LIN {X 0,Y 451.324,Z 462.44,A -85,B 0,C 180,E1 7902.427,E2 7902.427} C_VEL
LIN {X 0,Y 451.37,Z 462.44,A -85,B 0,C 180,E1 7908.389,E2 7908.389} C_VEL
LIN {X 0,Y 451.756,Z 462.44,A -85,B 0,C 180,E1 7914.229,E2 7914.229} C_VEL
LIN {X 0,Y 451.885,Z 462.44,A -85,B 0,C 180,E1 7919.999,E2 7919.999} C_VEL
LIN {X 0,Y 451.669,Z 462.44,A -85,B 0,C 180,E1 7925.77,E2 7925.77} C_VEL
LIN {X 0,Y 451.467,Z 462.44,A -85,B 0,C 180,E1 7931.606,E2 7931.606} C_VEL
LIN {X 0,Y 451.314,Z 462.44,A -85,B 0,C 180,E1 7937.571,E2 7937.571} C_VEL
LIN {X 0,Y 451.124,Z 462.44,A -85,B 0,C 180,E1 7943.747,E2 7943.747} C_VEL
LIN {X 0,Y 450.99,Z 462.44,A -85,B 0,C 180,E1 7950.233,E2 7950.233} C_VEL
LIN {X 0,Y 450.932,Z 462.44,A -85,B 0,C 180,E1 7957.179,E2 7957.179} C_VEL
LIN {X 0,Y 450.718,Z 462.44,A -85,B 0,C 180,E1 7962.348,E2 7962.348} C_VEL
LIN {X 0,Y 450.818,Z 463.134,A -85,B 0,C 180,E1 7967.336,E2 7967.336} C_VEL
LIN {X 0,Y 453.731,Z 468.536,A -85,B 0,C 180,E1 7967.816,E2 7967.816} C_VEL
LIN {X 0,Y 478.201,Z 510.738,A -85,B 0,C 180,E1 7971.496,E2 7971.496} C_VEL
LIN {X 0,Y 480.263,Z 516.821,A -85,B 0,C 180,E1 7971.862,E2 7971.862} C_VEL
LIN {X 0,Y 477.435,Z 558.442,A -85,B 0,C 180,E1 7973.15,E2 7973.15} C_VEL
LIN {X 0,Y 473.23,Z 596.553,A -85,B 0,C 180,E1 7975.116,E2 7975.116} C_VEL
LIN {X 0,Y 468.283,Z 632.377,A -85,B 0,C 180,E1 7977.816,E2 7977.816} C_VEL
LIN {X 0,Y 463.277,Z 664.621,A -85,B 0,C 180,E1 7981.141,E2 7981.141} C_VEL
LIN {X 0,Y 458.653,Z 694.094,A -85,B 0,C 180,E1 7985.206,E2 7985.206} C_VEL
LIN {X 0,Y 455.301,Z 719.108,A -85,B 0,C 180,E1 7989.817,E2 7989.817} C_VEL
LIN {X 0,Y 453.406,Z 738.227,A -85,B 0,C 180,E1 7994.505,E2 7994.505} C_VEL
LIN {X 0,Y 452.474,Z 752.113,A -85,B 0,C 180,E1 7999.394,E2 7999.394} C_VEL
LIN {X 0,Y 452.109,Z 760.491,A -85,B 0,C 180,E1 8004.234,E2 8004.234} C_VEL
LIN {X 0,Y 451.991,Z 763.61,A -85,B 0,C 180,E1 8008.08,E2 8008.08} C_VEL
LIN {X 0,Y 452.127,Z 763.56,A -85,B 0,C 180,E1 8011.919,E2 8011.919} C_VEL
LIN {X 0,Y 452.166,Z 759.161,A -85,B 0,C 180,E1 8016.731,E2 8016.731} C_VEL
LIN {X 0,Y 452.598,Z 749.606,A -85,B 0,C 180,E1 8021.579,E2 8021.579} C_VEL
LIN {X 0,Y 453.789,Z 734.435,A -85,B 0,C 180,E1 8026.476,E2 8026.476} C_VEL
LIN {X 0,Y 456.118,Z 712.614,A -85,B 0,C 180,E1 8031.417,E2 8031.417} C_VEL
LIN {X 0,Y 459.639,Z 688.185,A -85,B 0,C 180,E1 8035.618,E2 8035.618} C_VEL
LIN {X 0,Y 464.335,Z 657.713,A -85,B 0,C 180,E1 8039.57,E2 8039.57} C_VEL
LIN {X 0,Y 469.179,Z 625.711,A -85,B 0,C 180,E1 8042.671,E2 8042.671} C_VEL
LIN {X 0,Y 474.084,Z 589.727,A -85,B 0,C 180,E1 8045.202,E2 8045.202} C_VEL
LIN {X 0,Y 477.97,Z 553.189,A -85,B 0,C 180,E1 8046.954,E2 8046.954} C_VEL
LIN {X 0,Y 479.9,Z 515.284,A -85,B 0,C 180,E1 8048.123,E2 8048.123} C_VEL
LIN {X 0,Y 466.753,Z 490.221,A -85,B 0,C 180,E1 8050.103,E2 8050.103} C_VEL
LIN {X 0,Y 450.925,Z 463.373,A -85,B 0,C 180,E1 8052.551,E2 8052.551} C_VEL
LIN {X 0,Y 450.855,Z 462.44,A -85,B 0,C 180,E1 8052.815,E2 8052.815} C_VEL
LIN {X 0,Y 450.818,Z 462.44,A -85,B 0,C 180,E1 8057.807,E2 8057.807} C_VEL
LIN {X 0,Y 450.853,Z 462.44,A -85,B 0,C 180,E1 8063.708,E2 8063.708} C_VEL
LIN {X 0,Y 450.941,Z 462.44,A -85,B 0,C 180,E1 8069.763,E2 8069.763} C_VEL
LIN {X 0,Y 451.159,Z 462.44,A -85,B 0,C 180,E1 8076.255,E2 8076.255} C_VEL
LIN {X 0,Y 451.403,Z 462.44,A -85,B 0,C 180,E1 8082.432,E2 8082.432} C_VEL
LIN {X 0,Y 451.539,Z 462.44,A -85,B 0,C 180,E1 8088.396,E2 8088.396} C_VEL
LIN {X 0,Y 451.683,Z 462.44,A -85,B 0,C 180,E1 8094.23,E2 8094.23} C_VEL
LIN {X 0,Y 451.967,Z 462.44,A -85,B 0,C 180,E1 8100.001,E2 8100.001} C_VEL
LIN {X 0,Y 451.76,Z 462.44,A -85,B 0,C 180,E1 8105.771,E2 8105.771} C_VEL
LIN {X 0,Y 451.497,Z 462.44,A -85,B 0,C 180,E1 8111.608,E2 8111.608} C_VEL
LIN {X 0,Y 451.315,Z 462.44,A -85,B 0,C 180,E1 8117.573,E2 8117.573} C_VEL
LIN {X 0,Y 451.18,Z 462.44,A -85,B 0,C 180,E1 8123.746,E2 8123.746} C_VEL
LIN {X 0,Y 450.955,Z 462.44,A -85,B 0,C 180,E1 8130.238,E2 8130.238} C_VEL
LIN {X 0,Y 450.905,Z 462.44,A -85,B 0,C 180,E1 8137.185,E2 8137.185} C_VEL
LIN {X 0,Y 450.912,Z 462.534,A -85,B 0,C 180,E1 8142.762,E2 8142.762} C_VEL
LIN {X 0,Y 453.355,Z 468.115,A -85,B 0,C 180,E1 8143.193,E2 8143.193} C_VEL
LIN {X 0,Y 471.571,Z 501.672,A -85,B 0,C 180,E1 8146.001,E2 8146.001} C_VEL
LIN {X 0,Y 482.411,Z 522.561,A -85,B 0,C 180,E1 8147.593,E2 8147.593} C_VEL
LIN {X 0,Y 479.545,Z 563.603,A -85,B 0,C 180,E1 8148.943,E2 8148.943} C_VEL
LIN {X 0,Y 475.541,Z 604.001,A -85,B 0,C 180,E1 8150.986,E2 8150.986} C_VEL
LIN {X 0,Y 470.314,Z 619.687,A -85,B 0,C 180,E1 8151.742,E2 8151.742} C_VEL
LIN {X 0,Y 465.033,Z 634.714,A -85,B 0,C 180,E1 8152.6,E2 8152.6} C_VEL
LIN {X 0,Y 460.033,Z 668.804,A -85,B 0,C 180,E1 8155.687,E2 8155.687} C_VEL
LIN {X 0,Y 454.871,Z 702.031,A -85,B 0,C 180,E1 8159.647,E2 8159.647} C_VEL
LIN {X 0,Y 450.763,Z 729.018,A -85,B 0,C 180,E1 8163.904,E2 8163.904} C_VEL
LIN {X 0,Y 447.283,Z 753.133,A -85,B 0,C 180,E1 8168.993,E2 8168.993} C_VEL
LIN {X 0,Y 445.342,Z 771.29,A -85,B 0,C 180,E1 8174.217,E2 8174.217} C_VEL
LIN {X 0,Y 444.444,Z 783.404,A -85,B 0,C 180,E1 8179.2,E2 8179.2} C_VEL
LIN {X 0,Y 444.229,Z 790.904,A -85,B 0,C 180,E1 8184.131,E2 8184.131} C_VEL
LIN {X 0,Y 444.237,Z 793.657,A -85,B 0,C 180,E1 8188.047,E2 8188.047} C_VEL
LIN {X 0,Y 444.103,Z 793.657,A -85,B 0,C 180,E1 8191.954,E2 8191.954} C_VEL
LIN {X 0,Y 444.261,Z 789.703,A -85,B 0,C 180,E1 8196.851,E2 8196.851} C_VEL
LIN {X 0,Y 444.581,Z 781.433,A -85,B 0,C 180,E1 8201.791,E2 8201.791} C_VEL
LIN {X 0,Y 445.808,Z 766.683,A -85,B 0,C 180,E1 8207.288,E2 8207.288} C_VEL
LIN {X 0,Y 448.364,Z 745.171,A -85,B 0,C 180,E1 8212.852,E2 8212.852} C_VEL
LIN {X 0,Y 452.392,Z 718.357,A -85,B 0,C 180,E1 8217.942,E2 8217.942} C_VEL
LIN {X 0,Y 457.214,Z 687.111,A -85,B 0,C 180,E1 8222.272,E2 8222.272} C_VEL
LIN {X 0,Y 462.621,Z 651.579,A -85,B 0,C 180,E1 8225.989,E2 8225.989} C_VEL
LIN {X 0,Y 467.835,Z 613.132,A -85,B 0,C 180,E1 8228.969,E2 8228.969} C_VEL
LIN {X 0,Y 472.541,Z 571.788,A -85,B 0,C 180,E1 8231.253,E2 8231.253} C_VEL
LIN {X 0,Y 475.934,Z 530.855,A -85,B 0,C 180,E1 8232.745,E2 8232.745} C_VEL
LIN {X 0,Y 475.435,Z 524.554,A -85,B 0,C 180,E1 8232.994,E2 8232.994} C_VEL
LIN {X 0,Y 451.73,Z 478.738,A -85,B 0,C 180,E1 8236.767,E2 8236.767} C_VEL
LIN {X 0,Y 443.003,Z 463.385,A -85,B 0,C 180,E1 8238.243,E2 8238.243} C_VEL
LIN {X 0,Y 442.931,Z 462.44,A -85,B 0,C 180,E1 8238.357,E2 8238.357} C_VEL
LIN {X 0,Y 442.972,Z 462.44,A -85,B 0,C 180,E1 8245.12,E2 8245.12} C_VEL
LIN {X 0,Y 443.063,Z 462.44,A -85,B 0,C 180,E1 8251.419,E2 8251.419} C_VEL
LIN {X 0,Y 443.292,Z 462.44,A -85,B 0,C 180,E1 8257.933,E2 8257.933} C_VEL
LIN {X 0,Y 443.351,Z 462.44,A -85,B 0,C 180,E1 8264.145,E2 8264.145} C_VEL
LIN {X 0,Y 443.534,Z 462.44,A -85,B 0,C 180,E1 8270.172,E2 8270.172} C_VEL
LIN {X 0,Y 443.831,Z 462.44,A -85,B 0,C 180,E1 8276.087,E2 8276.087} C_VEL
LIN {X 0,Y 443.909,Z 462.44,A -85,B 0,C 180,E1 8281.953,E2 8281.953} C_VEL
LIN {X 0,Y 443.678,Z 462.44,A -85,B 0,C 180,E1 8288.239,E2 8288.239} C_VEL
LIN {X 0,Y 443.496,Z 462.44,A -85,B 0,C 180,E1 8293.824,E2 8293.824} C_VEL
LIN {X 0,Y 443.344,Z 462.44,A -85,B 0,C 180,E1 8299.966,E2 8299.966} C_VEL
LIN {X 0,Y 443.11,Z 462.44,A -85,B 0,C 180,E1 8306.369,E2 8306.369} C_VEL
LIN {X 0,Y 443.039,Z 462.44,A -85,B 0,C 180,E1 8313.143,E2 8313.143} C_VEL
LIN {X 0,Y 442.917,Z 462.44,A -85,B 0,C 180,E1 8318.162,E2 8318.162} C_VEL
LIN {X 0,Y 442.717,Z 462.44,A -85,B 0,C 180,E1 8324.092,E2 8324.092} C_VEL
LIN {X 0,Y 442.884,Z 462.44,A -85,B 0,C 180,E1 8326.27,E2 8326.27} C_VEL
LIN {X 0,Y 445.22,Z 468.052,A -85,B 0,C 180,E1 8326.71,E2 8326.71} C_VEL
LIN {X 0,Y 472.245,Z 513.43,A -85,B 0,C 180,E1 8330.901,E2 8330.901} C_VEL
LIN {X 0,Y 474.363,Z 518.736,A -85,B 0,C 180,E1 8331.263,E2 8331.263} C_VEL
LIN {X 0,Y 471.424,Z 559.474,A -85,B 0,C 180,E1 8332.543,E2 8332.543} C_VEL
LIN {X 0,Y 467.212,Z 596.323,A -85,B 0,C 180,E1 8334.457,E2 8334.457} C_VEL
LIN {X 0,Y 462.142,Z 631.059,A -85,B 0,C 180,E1 8337.07,E2 8337.07} C_VEL
LIN {X 0,Y 456.659,Z 663.805,A -85,B 0,C 180,E1 8340.448,E2 8340.448} C_VEL
LIN {X 0,Y 451.8,Z 692.62,A -85,B 0,C 180,E1 8344.436,E2 8344.436} C_VEL
LIN {X 0,Y 448.042,Z 717.186,A -85,B 0,C 180,E1 8348.957,E2 8348.957} C_VEL
LIN {X 0,Y 445.78,Z 736.484,A -85,B 0,C 180,E1 8353.727,E2 8353.727} C_VEL
LIN {X 0,Y 444.681,Z 750.963,A -85,B 0,C 180,E1 8358.709,E2 8358.709} C_VEL
LIN {X 0,Y 444.287,Z 759.281,A -85,B 0,C 180,E1 8363.149,E2 8363.149} C_VEL
LIN {X 0,Y 444.087,Z 763.61,A -85,B 0,C 180,E1 8368.046,E2 8368.046} C_VEL
LIN {X 0,Y 444.22,Z 763.56,A -85,B 0,C 180,E1 8371.953,E2 8371.953} C_VEL
LIN {X 0,Y 444.285,Z 759.162,A -85,B 0,C 180,E1 8376.851,E2 8376.851} C_VEL
LIN {X 0,Y 444.753,Z 749.609,A -85,B 0,C 180,E1 8381.787,E2 8381.787} C_VEL
LIN {X 0,Y 446.043,Z 734.439,A -85,B 0,C 180,E1 8386.771,E2 8386.771} C_VEL
LIN {X 0,Y 448.632,Z 713.182,A -85,B 0,C 180,E1 8391.793,E2 8391.793} C_VEL
LIN {X 0,Y 452.698,Z 687.251,A -85,B 0,C 180,E1 8396.306,E2 8396.306} C_VEL
LIN {X 0,Y 457.397,Z 659.179,A -85,B 0,C 180,E1 8400.005,E2 8400.005} C_VEL
LIN {X 0,Y 462.787,Z 626.357,A -85,B 0,C 180,E1 8403.249,E2 8403.249} C_VEL
LIN {X 0,Y 467.896,Z 590.924,A -85,B 0,C 180,E1 8405.78,E2 8405.78} C_VEL
LIN {X 0,Y 471.995,Z 554.466,A -85,B 0,C 180,E1 8407.554,E2 8407.554} C_VEL
LIN {X 0,Y 473.868,Z 517.772,A -85,B 0,C 180,E1 8408.729,E2 8408.729} C_VEL
LIN {X 0,Y 458.558,Z 489.802,A -85,B 0,C 180,E1 8411.071,E2 8411.071} C_VEL
LIN {X 0,Y 443.192,Z 464.273,A -85,B 0,C 180,E1 8413.545,E2 8413.545} C_VEL
LIN {X 0,Y 442.971,Z 462.44,A -85,B 0,C 180,E1 8413.673,E2 8413.673} C_VEL
LIN {X 0,Y 442.85,Z 462.44,A -85,B 0,C 180,E1 8419.494,E2 8419.494} C_VEL
LIN {X 0,Y 442.941,Z 462.44,A -85,B 0,C 180,E1 8425.126,E2 8425.126} C_VEL
LIN {X 0,Y 443.05,Z 462.44,A -85,B 0,C 180,E1 8431.421,E2 8431.421} C_VEL
LIN {X 0,Y 443.284,Z 462.44,A -85,B 0,C 180,E1 8437.935,E2 8437.935} C_VEL
LIN {X 0,Y 443.527,Z 462.44,A -85,B 0,C 180,E1 8444.154,E2 8444.154} C_VEL
LIN {X 0,Y 443.717,Z 462.44,A -85,B 0,C 180,E1 8450.178,E2 8450.178} C_VEL
LIN {X 0,Y 443.982,Z 462.44,A -85,B 0,C 180,E1 8456.091,E2 8456.091} C_VEL
LIN {X 0,Y 444.082,Z 462.44,A -85,B 0,C 180,E1 8461.955,E2 8461.955} C_VEL
LIN {X 0,Y 443.684,Z 462.44,A -85,B 0,C 180,E1 8468.244,E2 8468.244} C_VEL
LIN {X 0,Y 443.503,Z 462.44,A -85,B 0,C 180,E1 8473.826,E2 8473.826} C_VEL
LIN {X 0,Y 443.352,Z 462.44,A -85,B 0,C 180,E1 8479.968,E2 8479.968} C_VEL
LIN {X 0,Y 443.169,Z 462.44,A -85,B 0,C 180,E1 8486.367,E2 8486.367} C_VEL
LIN {X 0,Y 442.97,Z 462.44,A -85,B 0,C 180,E1 8493.152,E2 8493.152} C_VEL
LIN {X 0,Y 442.927,Z 462.44,A -85,B 0,C 180,E1 8498.164,E2 8498.164} C_VEL
LIN {X 0,Y 442.941,Z 462.44,A -85,B 0,C 180,E1 8501.703,E2 8501.703} C_VEL
LIN {X 0,Y 445.494,Z 468.203,A -85,B 0,C 180,E1 8502.203,E2 8502.203} C_VEL
LIN {X 0,Y 464.389,Z 502.201,A -85,B 0,C 180,E1 8505.244,E2 8505.244} C_VEL
LIN {X 0,Y 476.061,Z 525.75,A -85,B 0,C 180,E1 8507.1,E2 8507.1} C_VEL
LIN {X 0,Y 472.613,Z 569.283,A -85,B 0,C 180,E1 8508.627,E2 8508.627} C_VEL
LIN {X 0,Y 468.042,Z 610.25,A -85,B 0,C 180,E1 8510.838,E2 8510.838} C_VEL
LIN {X 0,Y 465.033,Z 634.714,A -85,B 0,C 180,E1 8512.6,E2 8512.6} C_VEL
LIN {X 0,Y 459.413,Z 649.427,A -85,B 0,C 180,E1 8513.567,E2 8513.567} C_VEL
LIN {X 0,Y 453.8,Z 663.557,A -85,B 0,C 180,E1 8514.649,E2 8514.649} C_VEL
LIN {X 0,Y 448.225,Z 698.38,A -85,B 0,C 180,E1 8518.709,E2 8518.709} C_VEL
LIN {X 0,Y 443.415,Z 728.161,A -85,B 0,C 180,E1 8523.317,E2 8523.317} C_VEL
LIN {X 0,Y 439.864,Z 751.939,A -85,B 0,C 180,E1 8528.329,E2 8528.329} C_VEL
LIN {X 0,Y 437.727,Z 769.757,A -85,B 0,C 180,E1 8533.419,E2 8533.419} C_VEL
LIN {X 0,Y 436.714,Z 781.432,A -85,B 0,C 180,E1 8537.993,E2 8537.993} C_VEL
LIN {X 0,Y 436.333,Z 789.702,A -85,B 0,C 180,E1 8543.024,E2 8543.024} C_VEL
LIN {X 0,Y 436.342,Z 793.657,A -85,B 0,C 180,E1 8548.011,E2 8548.011} C_VEL
LIN {X 0,Y 436.221,Z 793.657,A -85,B 0,C 180,E1 8551.989,E2 8551.989} C_VEL
LIN {X 0,Y 436.359,Z 789.703,A -85,B 0,C 180,E1 8556.976,E2 8556.976} C_VEL
LIN {X 0,Y 436.716,Z 781.433,A -85,B 0,C 180,E1 8562.007,E2 8562.007} C_VEL
LIN {X 0,Y 438.069,Z 766.684,A -85,B 0,C 180,E1 8567.604,E2 8567.604} C_VEL
LIN {X 0,Y 440.765,Z 745.169,A -85,B 0,C 180,E1 8573.269,E2 8573.269} C_VEL
LIN {X 0,Y 444.538,Z 721.031,A -85,B 0,C 180,E1 8577.903,E2 8577.903} C_VEL
LIN {X 0,Y 449.665,Z 689.377,A -85,B 0,C 180,E1 8582.456,E2 8582.456} C_VEL
LIN {X 0,Y 455.236,Z 654.657,A -85,B 0,C 180,E1 8586.207,E2 8586.207} C_VEL
LIN {X 0,Y 460.836,Z 615.843,A -85,B 0,C 180,E1 8589.321,E2 8589.321} C_VEL
LIN {X 0,Y 465.673,Z 575.86,A -85,B 0,C 180,E1 8591.625,E2 8591.625} C_VEL
LIN {X 0,Y 469.242,Z 536.544,A -85,B 0,C 180,E1 8593.174,E2 8593.174} C_VEL
LIN {X 0,Y 469.142,Z 527.516,A -85,B 0,C 180,E1 8593.525,E2 8593.525} C_VEL
LIN {X 0,Y 447.151,Z 484.199,A -85,B 0,C 180,E1 8597.212,E2 8597.212} C_VEL
LIN {X 0,Y 435.266,Z 464.439,A -85,B 0,C 180,E1 8599.273,E2 8599.273} C_VEL
LIN {X 0,Y 435.031,Z 462.44,A -85,B 0,C 180,E1 8599.519,E2 8599.519} C_VEL
LIN {X 0,Y 435.066,Z 462.44,A -85,B 0,C 180,E1 8606.643,E2 8606.643} C_VEL
LIN {X 0,Y 435.214,Z 462.44,A -85,B 0,C 180,E1 8613.112,E2 8613.112} C_VEL
LIN {X 0,Y 435.486,Z 462.44,A -85,B 0,C 180,E1 8619.844,E2 8619.844} C_VEL
LIN {X 0,Y 435.443,Z 462.44,A -85,B 0,C 180,E1 8626.811,E2 8626.811} C_VEL
LIN {X 0,Y 435.809,Z 462.44,A -85,B 0,C 180,E1 8632.011,E2 8632.011} C_VEL
LIN {X 0,Y 436.195,Z 462.44,A -85,B 0,C 180,E1 8638.01,E2 8638.01} C_VEL
LIN {X 0,Y 435.965,Z 462.44,A -85,B 0,C 180,E1 8643.981,E2 8643.981} C_VEL
LIN {X 0,Y 435.74,Z 462.44,A -85,B 0,C 180,E1 8650.003,E2 8650.003} C_VEL
LIN {X 0,Y 435.527,Z 462.44,A -85,B 0,C 180,E1 8656.145,E2 8656.145} C_VEL
LIN {X 0,Y 435.314,Z 462.44,A -85,B 0,C 180,E1 8662.491,E2 8662.491} C_VEL
LIN {X 0,Y 435.066,Z 462.44,A -85,B 0,C 180,E1 8669.534,E2 8669.534} C_VEL
LIN {X 0,Y 435.106,Z 462.44,A -85,B 0,C 180,E1 8673.828,E2 8673.828} C_VEL
LIN {X 0,Y 434.894,Z 462.44,A -85,B 0,C 180,E1 8680.008,E2 8680.008} C_VEL
LIN {X 0,Y 434.855,Z 462.44,A -85,B 0,C 180,E1 8685.149,E2 8685.149} C_VEL
LIN {X 0,Y 437.294,Z 468.096,A -85,B 0,C 180,E1 8685.634,E2 8685.634} C_VEL
LIN {X 0,Y 464.383,Z 512.958,A -85,B 0,C 180,E1 8690.006,E2 8690.006} C_VEL
LIN {X 0,Y 468.332,Z 521.89,A -85,B 0,C 180,E1 8690.691,E2 8690.691} C_VEL
LIN {X 0,Y 465.319,Z 560.942,A -85,B 0,C 180,E1 8691.959,E2 8691.959} C_VEL
LIN {X 0,Y 460.918,Z 597.783,A -85,B 0,C 180,E1 8693.896,E2 8693.896} C_VEL
LIN {X 0,Y 455.814,Z 631.227,A -85,B 0,C 180,E1 8696.436,E2 8696.436} C_VEL
LIN {X 0,Y 449.976,Z 663.864,A -85,B 0,C 180,E1 8699.839,E2 8699.839} C_VEL
LIN {X 0,Y 444.622,Z 693.348,A -85,B 0,C 180,E1 8703.992,E2 8703.992} C_VEL
LIN {X 0,Y 440.471,Z 718.108,A -85,B 0,C 180,E1 8708.667,E2 8708.667} C_VEL
LIN {X 0,Y 438.047,Z 736.785,A -85,B 0,C 180,E1 8713.431,E2 8713.431} C_VEL
LIN {X 0,Y 436.807,Z 750.961,A -85,B 0,C 180,E1 8718.503,E2 8718.503} C_VEL
LIN {X 0,Y 436.386,Z 759.28,A -85,B 0,C 180,E1 8723.025,E2 8723.025} C_VEL
LIN {X 0,Y 436.205,Z 763.61,A -85,B 0,C 180,E1 8728.011,E2 8728.011} C_VEL
LIN {X 0,Y 436.324,Z 763.56,A -85,B 0,C 180,E1 8731.989,E2 8731.989} C_VEL
LIN {X 0,Y 436.388,Z 759.163,A -85,B 0,C 180,E1 8736.975,E2 8736.975} C_VEL
LIN {X 0,Y 436.914,Z 749.61,A -85,B 0,C 180,E1 8742.001,E2 8742.001} C_VEL
LIN {X 0,Y 438.549,Z 732.978,A -85,B 0,C 180,E1 8747.584,E2 8747.584} C_VEL
LIN {X 0,Y 441.393,Z 712.485,A -85,B 0,C 180,E1 8752.435,E2 8752.435} C_VEL
LIN {X 0,Y 445.578,Z 688.037,A -85,B 0,C 180,E1 8756.76,E2 8756.76} C_VEL
LIN {X 0,Y 450.956,Z 658.375,A -85,B 0,C 180,E1 8760.716,E2 8760.716} C_VEL
LIN {X 0,Y 456.465,Z 626.604,A -85,B 0,C 180,E1 8763.88,E2 8763.88} C_VEL
LIN {X 0,Y 461.765,Z 591.606,A -85,B 0,C 180,E1 8766.393,E2 8766.393} C_VEL
LIN {X 0,Y 466.045,Z 554.605,A -85,B 0,C 180,E1 8768.196,E2 8768.196} C_VEL
LIN {X 0,Y 467.817,Z 520.484,A -85,B 0,C 180,E1 8769.318,E2 8769.318} C_VEL
LIN {X 0,Y 450.73,Z 489.836,A -85,B 0,C 180,E1 8772.031,E2 8772.031} C_VEL
LIN {X 0,Y 435.209,Z 464.327,A -85,B 0,C 180,E1 8774.646,E2 8774.646} C_VEL
LIN {X 0,Y 434.953,Z 462.44,A -85,B 0,C 180,E1 8774.879,E2 8774.879} C_VEL
LIN {X 0,Y 434.899,Z 462.44,A -85,B 0,C 180,E1 8781.201,E2 8781.201} C_VEL
LIN {X 0,Y 435.045,Z 462.44,A -85,B 0,C 180,E1 8786.647,E2 8786.647} C_VEL
LIN {X 0,Y 435.195,Z 462.44,A -85,B 0,C 180,E1 8793.114,E2 8793.114} C_VEL
LIN {X 0,Y 435.455,Z 462.44,A -85,B 0,C 180,E1 8799.855,E2 8799.855} C_VEL
LIN {X 0,Y 435.675,Z 462.44,A -85,B 0,C 180,E1 8805.923,E2 8805.923} C_VEL
LIN {X 0,Y 435.828,Z 462.44,A -85,B 0,C 180,E1 8812.014,E2 8812.014} C_VEL
LIN {X 0,Y 436.075,Z 462.44,A -85,B 0,C 180,E1 8818.012,E2 8818.012} C_VEL
LIN {X 0,Y 435.924,Z 462.44,A -85,B 0,C 180,E1 8823.984,E2 8823.984} C_VEL
LIN {X 0,Y 435.705,Z 462.44,A -85,B 0,C 180,E1 8830.006,E2 8830.006} C_VEL
LIN {X 0,Y 435.53,Z 462.44,A -85,B 0,C 180,E1 8836.147,E2 8836.147} C_VEL
LIN {X 0,Y 435.351,Z 462.44,A -85,B 0,C 180,E1 8842.492,E2 8842.492} C_VEL
LIN {X 0,Y 435.077,Z 462.44,A -85,B 0,C 180,E1 8849.156,E2 8849.156} C_VEL
LIN {X 0,Y 435.041,Z 462.44,A -85,B 0,C 180,E1 8853.836,E2 8853.836} C_VEL
LIN {X 0,Y 435.025,Z 463.003,A -85,B 0,C 180,E1 8860.664,E2 8860.664} C_VEL
LIN {X 0,Y 437.742,Z 468.392,A -85,B 0,C 180,E1 8861.174,E2 8861.174} C_VEL
LIN {X 0,Y 457.3,Z 502.951,A -85,B 0,C 180,E1 8864.461,E2 8864.461} C_VEL
LIN {X 0,Y 469.649,Z 529.883,A -85,B 0,C 180,E1 8866.61,E2 8866.61} C_VEL
LIN {X 0,Y 465.721,Z 574.382,A -85,B 0,C 180,E1 8868.291,E2 8868.291} C_VEL
LIN {X 0,Y 460.649,Z 616.24,A -85,B 0,C 180,E1 8870.695,E2 8870.695} C_VEL
LIN {X 0,Y 455.136,Z 654.78,A -85,B 0,C 180,E1 8873.799,E2 8873.799} C_VEL
LIN {X 0,Y 453.8,Z 663.557,A -85,B 0,C 180,E1 8874.649,E2 8874.649} C_VEL
LIN {X 0,Y 448.075,Z 677.236,A -85,B 0,C 180,E1 8875.848,E2 8875.848} C_VEL
LIN {X 0,Y 442.332,Z 690.195,A -85,B 0,C 180,E1 8877.178,E2 8877.178} C_VEL
LIN {X 0,Y 437.25,Z 720.049,A -85,B 0,C 180,E1 8881.529,E2 8881.529} C_VEL
LIN {X 0,Y 433.239,Z 746.212,A -85,B 0,C 180,E1 8886.575,E2 8886.575} C_VEL
LIN {X 0,Y 430.351,Z 767.046,A -85,B 0,C 180,E1 8892.193,E2 8892.193} C_VEL
LIN {X 0,Y 428.88,Z 781.432,A -85,B 0,C 180,E1 8897.771,E2 8897.771} C_VEL
LIN {X 0,Y 428.442,Z 789.702,A -85,B 0,C 180,E1 8902.895,E2 8902.895} C_VEL
LIN {X 0,Y 428.434,Z 793.657,A -85,B 0,C 180,E1 8907.975,E2 8907.975} C_VEL
LIN {X 0,Y 428.316,Z 793.657,A -85,B 0,C 180,E1 8912.026,E2 8912.026} C_VEL
LIN {X 0,Y 428.467,Z 789.703,A -85,B 0,C 180,E1 8917.105,E2 8917.105} C_VEL
LIN {X 0,Y 428.866,Z 781.432,A -85,B 0,C 180,E1 8922.23,E2 8922.23} C_VEL
LIN {X 0,Y 430.258,Z 767.139,A -85,B 0,C 180,E1 8927.779,E2 8927.779} C_VEL
LIN {X 0,Y 432.919,Z 747.323,A -85,B 0,C 180,E1 8933.17,E2 8933.17} C_VEL
LIN {X 0,Y 436.897,Z 722.099,A -85,B 0,C 180,E1 8938.114,E2 8938.114} C_VEL
LIN {X 0,Y 441.913,Z 692.562,A -85,B 0,C 180,E1 8942.514,E2 8942.514} C_VEL
LIN {X 0,Y 447.452,Z 659.789,A -85,B 0,C 180,E1 8946.218,E2 8946.218} C_VEL
LIN {X 0,Y 453.028,Z 623.693,A -85,B 0,C 180,E1 8949.316,E2 8949.316} C_VEL
LIN {X 0,Y 458.395,Z 583.756,A -85,B 0,C 180,E1 8951.827,E2 8951.827} C_VEL
LIN {X 0,Y 462.675,Z 542.504,A -85,B 0,C 180,E1 8953.616,E2 8953.616} C_VEL
LIN {X 0,Y 462.973,Z 530.68,A -85,B 0,C 180,E1 8954.056,E2 8954.056} C_VEL
LIN {X 0,Y 442.608,Z 489.616,A -85,B 0,C 180,E1 8957.667,E2 8957.667} C_VEL
LIN {X 0,Y 428.452,Z 466.917,A -85,B 0,C 180,E1 8960.19,E2 8960.19} C_VEL
LIN {X 0,Y 427.036,Z 462.44,A -85,B 0,C 180,E1 8960.593,E2 8960.593} C_VEL
LIN {X 0,Y 427.11,Z 462.44,A -85,B 0,C 180,E1 8967.879,E2 8967.879} C_VEL
LIN {X 0,Y 427.346,Z 462.44,A -85,B 0,C 180,E1 8974.84,E2 8974.84} C_VEL
LIN {X 0,Y 427.554,Z 462.44,A -85,B 0,C 180,E1 8981.415,E2 8981.415} C_VEL
LIN {X 0,Y 427.588,Z 462.44,A -85,B 0,C 180,E1 8987.733,E2 8987.733} C_VEL
LIN {X 0,Y 427.995,Z 462.44,A -85,B 0,C 180,E1 8993.907,E2 8993.907} C_VEL
LIN {X 0,Y 428.197,Z 462.44,A -85,B 0,C 180,E1 8999.999,E2 8999.999} C_VEL
LIN {X 0,Y 427.921,Z 462.44,A -85,B 0,C 180,E1 9006.092,E2 9006.092} C_VEL
LIN {X 0,Y 427.69,Z 462.44,A -85,B 0,C 180,E1 9012.261,E2 9012.261} C_VEL
LIN {X 0,Y 427.504,Z 462.44,A -85,B 0,C 180,E1 9018.585,E2 9018.585} C_VEL
LIN {X 0,Y 427.298,Z 462.44,A -85,B 0,C 180,E1 9025.16,E2 9025.16} C_VEL
LIN {X 0,Y 427.175,Z 462.44,A -85,B 0,C 180,E1 9032.113,E2 9032.113} C_VEL
LIN {X 0,Y 427.028,Z 462.44,A -85,B 0,C 180,E1 9038.734,E2 9038.734} C_VEL
LIN {X 0,Y 426.918,Z 462.623,A -85,B 0,C 180,E1 9044.002,E2 9044.002} C_VEL
LIN {X 0,Y 429.491,Z 468.277,A -85,B 0,C 180,E1 9044.517,E2 9044.517} C_VEL
LIN {X 0,Y 455.002,Z 510.014,A -85,B 0,C 180,E1 9048.833,E2 9048.833} C_VEL
LIN {X 0,Y 462.323,Z 523.77,A -85,B 0,C 180,E1 9050.07,E2 9050.07} C_VEL
LIN {X 0,Y 459.225,Z 562.268,A -85,B 0,C 180,E1 9051.362,E2 9051.362} C_VEL
LIN {X 0,Y 454.636,Z 598.86,A -85,B 0,C 180,E1 9053.316,E2 9053.316} C_VEL
LIN {X 0,Y 449.222,Z 632.796,A -85,B 0,C 180,E1 9055.925,E2 9055.925} C_VEL
LIN {X 0,Y 443.174,Z 664.771,A -85,B 0,C 180,E1 9059.313,E2 9059.313} C_VEL
LIN {X 0,Y 437.534,Z 693.715,A -85,B 0,C 180,E1 9063.47,E2 9063.47} C_VEL
LIN {X 0,Y 433.032,Z 718.344,A -85,B 0,C 180,E1 9068.203,E2 9068.203} C_VEL
LIN {X 0,Y 430.356,Z 737.217,A -85,B 0,C 180,E1 9073.126,E2 9073.126} C_VEL
LIN {X 0,Y 428.948,Z 751.205,A -85,B 0,C 180,E1 9078.289,E2 9078.289} C_VEL
LIN {X 0,Y 428.519,Z 759.291,A -85,B 0,C 180,E1 9082.896,E2 9082.896} C_VEL
LIN {X 0,Y 428.301,Z 763.609,A -85,B 0,C 180,E1 9087.974,E2 9087.974} C_VEL
LIN {X 0,Y 428.417,Z 763.56,A -85,B 0,C 180,E1 9092.025,E2 9092.025} C_VEL
LIN {X 0,Y 428.526,Z 759.179,A -85,B 0,C 180,E1 9097.104,E2 9097.104} C_VEL
LIN {X 0,Y 429.095,Z 749.899,A -85,B 0,C 180,E1 9102.223,E2 9102.223} C_VEL
LIN {X 0,Y 430.664,Z 735.252,A -85,B 0,C 180,E1 9107.388,E2 9107.388} C_VEL
LIN {X 0,Y 433.766,Z 714.39,A -85,B 0,C 180,E1 9112.58,E2 9112.58} C_VEL
LIN {X 0,Y 438.446,Z 689.08,A -85,B 0,C 180,E1 9117.196,E2 9117.196} C_VEL
LIN {X 0,Y 444.027,Z 660.394,A -85,B 0,C 180,E1 9121.127,E2 9121.127} C_VEL
LIN {X 0,Y 449.988,Z 627.779,A -85,B 0,C 180,E1 9124.436,E2 9124.436} C_VEL
LIN {X 0,Y 455.499,Z 592.959,A -85,B 0,C 180,E1 9126.963,E2 9126.963} C_VEL
LIN {X 0,Y 460.095,Z 554.477,A -85,B 0,C 180,E1 9128.86,E2 9128.86} C_VEL
LIN {X 0,Y 461.92,Z 523.43,A -85,B 0,C 180,E1 9129.895,E2 9129.895} C_VEL
LIN {X 0,Y 440.366,Z 485.239,A -85,B 0,C 180,E1 9133.476,E2 9133.476} C_VEL
LIN {X 0,Y 427.094,Z 463.471,A -85,B 0,C 180,E1 9135.852,E2 9135.852} C_VEL
LIN {X 0,Y 427.019,Z 462.44,A -85,B 0,C 180,E1 9135.983,E2 9135.983} C_VEL
LIN {X 0,Y 426.974,Z 462.44,A -85,B 0,C 180,E1 9142.932,E2 9142.932} C_VEL
LIN {X 0,Y 427.149,Z 462.44,A -85,B 0,C 180,E1 9150.252,E2 9150.252} C_VEL
LIN {X 0,Y 427.394,Z 462.44,A -85,B 0,C 180,E1 9157.088,E2 9157.088} C_VEL
LIN {X 0,Y 427.673,Z 462.44,A -85,B 0,C 180,E1 9163.55,E2 9163.55} C_VEL
LIN {X 0,Y 427.858,Z 462.44,A -85,B 0,C 180,E1 9169.811,E2 9169.811} C_VEL
LIN {X 0,Y 428.142,Z 462.44,A -85,B 0,C 180,E1 9175.946,E2 9175.946} C_VEL
LIN {X 0,Y 428.284,Z 462.44,A -85,B 0,C 180,E1 9182.027,E2 9182.027} C_VEL
LIN {X 0,Y 427.915,Z 462.44,A -85,B 0,C 180,E1 9188.137,E2 9188.137} C_VEL
LIN {X 0,Y 427.633,Z 462.44,A -85,B 0,C 180,E1 9194.35,E2 9194.35} C_VEL
LIN {X 0,Y 427.441,Z 462.44,A -85,B 0,C 180,E1 9200.745,E2 9200.745} C_VEL
LIN {X 0,Y 427.228,Z 462.44,A -85,B 0,C 180,E1 9207.622,E2 9207.622} C_VEL
LIN {X 0,Y 427.035,Z 462.44,A -85,B 0,C 180,E1 9214.56,E2 9214.56} C_VEL
LIN {X 0,Y 427.06,Z 462.44,A -85,B 0,C 180,E1 9219.466,E2 9219.466} C_VEL
LIN {X 0,Y 429.511,Z 468.152,A -85,B 0,C 180,E1 9220.005,E2 9220.005} C_VEL
LIN {X 0,Y 448.905,Z 501.013,A -85,B 0,C 180,E1 9223.407,E2 9223.407} C_VEL
LIN {X 0,Y 463.368,Z 532.549,A -85,B 0,C 180,E1 9226.061,E2 9226.061} C_VEL
LIN {X 0,Y 459.461,Z 573.807,A -85,B 0,C 180,E1 9227.66,E2 9227.66} C_VEL
LIN {X 0,Y 453.948,Z 616.443,A -85,B 0,C 180,E1 9230.154,E2 9230.154} C_VEL
LIN {X 0,Y 448.191,Z 654.816,A -85,B 0,C 180,E1 9233.29,E2 9233.29} C_VEL
LIN {X 0,Y 442.332,Z 690.195,A -85,B 0,C 180,E1 9237.178,E2 9237.178} C_VEL
LIN {X 0,Y 436.532,Z 702.603,A -85,B 0,C 180,E1 9238.621,E2 9238.621} C_VEL
LIN {X 0,Y 430.823,Z 714.268,A -85,B 0,C 180,E1 9240.168,E2 9240.168} C_VEL
LIN {X 0,Y 426.456,Z 739.464,A -85,B 0,C 180,E1 9244.782,E2 9244.782} C_VEL
LIN {X 0,Y 423.41,Z 759.559,A -85,B 0,C 180,E1 9249.594,E2 9249.594} C_VEL
LIN {X 0,Y 421.578,Z 775.425,A -85,B 0,C 180,E1 9254.907,E2 9254.907} C_VEL
LIN {X 0,Y 420.744,Z 785.329,A -85,B 0,C 180,E1 9259.634,E2 9259.634} C_VEL
LIN {X 0,Y 420.529,Z 790.904,A -85,B 0,C 180,E1 9263.799,E2 9263.799} C_VEL
LIN {X 0,Y 420.527,Z 793.657,A -85,B 0,C 180,E1 9267.937,E2 9267.937} C_VEL
LIN {X 0,Y 420.411,Z 793.657,A -85,B 0,C 180,E1 9272.064,E2 9272.064} C_VEL
LIN {X 0,Y 420.594,Z 789.703,A -85,B 0,C 180,E1 9277.238,E2 9277.238} C_VEL
LIN {X 0,Y 421.004,Z 781.432,A -85,B 0,C 180,E1 9282.462,E2 9282.462} C_VEL
LIN {X 0,Y 422.465,Z 767.488,A -85,B 0,C 180,E1 9287.995,E2 9287.995} C_VEL
LIN {X 0,Y 424.991,Z 749.047,A -85,B 0,C 180,E1 9293.073,E2 9293.073} C_VEL
LIN {X 0,Y 428.811,Z 725.494,A -85,B 0,C 180,E1 9297.927,E2 9297.927} C_VEL
LIN {X 0,Y 433.857,Z 697.629,A -85,B 0,C 180,E1 9302.306,E2 9302.306} C_VEL
LIN {X 0,Y 439.989,Z 663.06,A -85,B 0,C 180,E1 9306.415,E2 9306.415} C_VEL
LIN {X 0,Y 446.273,Z 624.611,A -85,B 0,C 180,E1 9309.821,E2 9309.821} C_VEL
LIN {X 0,Y 452.092,Z 584.176,A -85,B 0,C 180,E1 9312.433,E2 9312.433} C_VEL
LIN {X 0,Y 456.528,Z 543.828,A -85,B 0,C 180,E1 9314.221,E2 9314.221} C_VEL
LIN {X 0,Y 456.754,Z 533.797,A -85,B 0,C 180,E1 9314.612,E2 9314.612} C_VEL
LIN {X 0,Y 438.388,Z 495.436,A -85,B 0,C 180,E1 9318.084,E2 9318.084} C_VEL
LIN {X 0,Y 420.484,Z 466.801,A -85,B 0,C 180,E1 9321.404,E2 9321.404} C_VEL
LIN {X 0,Y 419.123,Z 462.44,A -85,B 0,C 180,E1 9321.793,E2 9321.793} C_VEL
LIN {X 0,Y 419.111,Z 462.44,A -85,B 0,C 180,E1 9327.189,E2 9327.189} C_VEL
LIN {X 0,Y 419.279,Z 462.44,A -85,B 0,C 180,E1 9332.003,E2 9332.003} C_VEL
LIN {X 0,Y 419.545,Z 462.44,A -85,B 0,C 180,E1 9338.846,E2 9338.846} C_VEL
LIN {X 0,Y 419.587,Z 462.44,A -85,B 0,C 180,E1 9345.369,E2 9345.369} C_VEL
LIN {X 0,Y 419.96,Z 462.44,A -85,B 0,C 180,E1 9351.708,E2 9351.708} C_VEL
LIN {X 0,Y 420.368,Z 462.44,A -85,B 0,C 180,E1 9357.935,E2 9357.935} C_VEL
LIN {X 0,Y 420.139,Z 462.44,A -85,B 0,C 180,E1 9364.132,E2 9364.132} C_VEL
LIN {X 0,Y 419.869,Z 462.44,A -85,B 0,C 180,E1 9370.385,E2 9370.385} C_VEL
LIN {X 0,Y 419.657,Z 462.44,A -85,B 0,C 180,E1 9376.773,E2 9376.773} C_VEL
LIN {X 0,Y 419.393,Z 462.44,A -85,B 0,C 180,E1 9383.395,E2 9383.395} C_VEL
LIN {X 0,Y 419.237,Z 462.44,A -85,B 0,C 180,E1 9390.368,E2 9390.368} C_VEL
LIN {X 0,Y 419.129,Z 462.44,A -85,B 0,C 180,E1 9397.367,E2 9397.367} C_VEL
LIN {X 0,Y 419.009,Z 462.484,A -85,B 0,C 180,E1 9402.766,E2 9402.766} C_VEL
LIN {X 0,Y 421.357,Z 468.036,A -85,B 0,C 180,E1 9403.273,E2 9403.273} C_VEL
LIN {X 0,Y 443.986,Z 504.154,A -85,B 0,C 180,E1 9407.31,E2 9407.31} C_VEL
LIN {X 0,Y 456.386,Z 527.93,A -85,B 0,C 180,E1 9409.511,E2 9409.511} C_VEL
LIN {X 0,Y 452.688,Z 567.652,A -85,B 0,C 180,E1 9410.929,E2 9410.929} C_VEL
LIN {X 0,Y 447.218,Z 607.227,A -85,B 0,C 180,E1 9413.213,E2 9413.213} C_VEL
LIN {X 0,Y 440.948,Z 642.781,A -85,B 0,C 180,E1 9416.215,E2 9416.215} C_VEL
LIN {X 0,Y 434.573,Z 674.587,A -85,B 0,C 180,E1 9419.944,E2 9419.944} C_VEL
LIN {X 0,Y 428.924,Z 701.44,A -85,B 0,C 180,E1 9424.206,E2 9424.206} C_VEL
LIN {X 0,Y 424.679,Z 724.425,A -85,B 0,C 180,E1 9429.112,E2 9429.112} C_VEL
LIN {X 0,Y 422.105,Z 742.429,A -85,B 0,C 180,E1 9434.393,E2 9434.393} C_VEL
LIN {X 0,Y 420.963,Z 754.684,A -85,B 0,C 180,E1 9439.639,E2 9439.639} C_VEL
LIN {X 0,Y 420.545,Z 760.774,A -85,B 0,C 180,E1 9443.799,E2 9443.799} C_VEL
LIN {X 0,Y 420.399,Z 763.807,A -85,B 0,C 180,E1 9447.936,E2 9447.936} C_VEL
LIN {X 0,Y 420.513,Z 763.757,A -85,B 0,C 180,E1 9452.064,E2 9452.064} C_VEL
LIN {X 0,Y 420.653,Z 759.494,A -85,B 0,C 180,E1 9457.238,E2 9457.238} C_VEL
LIN {X 0,Y 421.412,Z 749.229,A -85,B 0,C 180,E1 9462.903,E2 9462.903} C_VEL
LIN {X 0,Y 423.241,Z 734.004,A -85,B 0,C 180,E1 9468.224,E2 9468.224} C_VEL
LIN {X 0,Y 426.837,Z 712.496,A -85,B 0,C 180,E1 9473.52,E2 9473.52} C_VEL
LIN {X 0,Y 431.95,Z 686.863,A -85,B 0,C 180,E1 9478.165,E2 9478.165} C_VEL
LIN {X 0,Y 437.822,Z 658.541,A -85,B 0,C 180,E1 9481.991,E2 9481.991} C_VEL
LIN {X 0,Y 443.893,Z 626.509,A -85,B 0,C 180,E1 9485.192,E2 9485.192} C_VEL
LIN {X 0,Y 449.602,Z 590.998,A -85,B 0,C 180,E1 9487.748,E2 9487.748} C_VEL
LIN {X 0,Y 454.328,Z 552.898,A -85,B 0,C 180,E1 9489.591,E2 9489.591} C_VEL
LIN {X 0,Y 455.986,Z 526.459,A -85,B 0,C 180,E1 9490.491,E2 9490.491} C_VEL
LIN {X 0,Y 432.791,Z 485.535,A -85,B 0,C 180,E1 9494.517,E2 9494.517} C_VEL
LIN {X 0,Y 420.34,Z 466.699,A -85,B 0,C 180,E1 9496.819,E2 9496.819} C_VEL
LIN {X 0,Y 419.084,Z 462.44,A -85,B 0,C 180,E1 9497.154,E2 9497.154} C_VEL
LIN {X 0,Y 419.084,Z 462.44,A -85,B 0,C 180,E1 9504.691,E2 9504.691} C_VEL
LIN {X 0,Y 419.263,Z 462.44,A -85,B 0,C 180,E1 9512.004,E2 9512.004} C_VEL
LIN {X 0,Y 419.536,Z 462.44,A -85,B 0,C 180,E1 9518.848,E2 9518.848} C_VEL
LIN {X 0,Y 419.812,Z 462.44,A -85,B 0,C 180,E1 9525.379,E2 9525.379} C_VEL
LIN {X 0,Y 419.992,Z 462.44,A -85,B 0,C 180,E1 9531.711,E2 9531.711} C_VEL
LIN {X 0,Y 420.264,Z 462.44,A -85,B 0,C 180,E1 9537.937,E2 9537.937} C_VEL
LIN {X 0,Y 420.111,Z 462.44,A -85,B 0,C 180,E1 9544.134,E2 9544.134} C_VEL
LIN {X 0,Y 419.848,Z 462.44,A -85,B 0,C 180,E1 9550.388,E2 9550.388} C_VEL
LIN {X 0,Y 419.664,Z 462.44,A -85,B 0,C 180,E1 9556.776,E2 9556.776} C_VEL
LIN {X 0,Y 419.448,Z 462.44,A -85,B 0,C 180,E1 9563.394,E2 9563.394} C_VEL
LIN {X 0,Y 419.217,Z 462.44,A -85,B 0,C 180,E1 9570.372,E2 9570.372} C_VEL
LIN {X 0,Y 419.112,Z 462.44,A -85,B 0,C 180,E1 9577.364,E2 9577.364} C_VEL
LIN {X 0,Y 419.121,Z 462.44,A -85,B 0,C 180,E1 9578.261,E2 9578.261} C_VEL
LIN {X 0,Y 421.538,Z 468.055,A -85,B 0,C 180,E1 9578.803,E2 9578.803} C_VEL
LIN {X 0,Y 441.46,Z 501.105,A -85,B 0,C 180,E1 9582.469,E2 9582.469} C_VEL
LIN {X 0,Y 457.135,Z 536.043,A -85,B 0,C 180,E1 9585.524,E2 9585.524} C_VEL
LIN {X 0,Y 452.917,Z 576.959,A -85,B 0,C 180,E1 9587.191,E2 9587.191} C_VEL
LIN {X 0,Y 447.306,Z 616.781,A -85,B 0,C 180,E1 9589.588,E2 9589.588} C_VEL
LIN {X 0,Y 441.236,Z 655.05,A -85,B 0,C 180,E1 9592.784,E2 9592.784} C_VEL
LIN {X 0,Y 435.313,Z 689.25,A -85,B 0,C 180,E1 9596.585,E2 9596.585} C_VEL
LIN {X 0,Y 430.823,Z 714.268,A -85,B 0,C 180,E1 9600.168,E2 9600.168} C_VEL
LIN {X 0,Y 425.183,Z 725.309,A -85,B 0,C 180,E1 9601.838,E2 9601.838} C_VEL
LIN {X 0,Y 419.596,Z 735.594,A -85,B 0,C 180,E1 9603.607,E2 9603.607} C_VEL
LIN {X 0,Y 415.86,Z 758.074,A -85,B 0,C 180,E1 9608.928,E2 9608.928} C_VEL
LIN {X 0,Y 413.923,Z 774.026,A -85,B 0,C 180,E1 9614.077,E2 9614.077} C_VEL
LIN {X 0,Y 412.865,Z 785.329,A -85,B 0,C 180,E1 9619.434,E2 9619.434} C_VEL
LIN {X 0,Y 412.629,Z 790.904,A -85,B 0,C 180,E1 9623.68,E2 9623.68} C_VEL
LIN {X 0,Y 412.619,Z 793.657,A -85,B 0,C 180,E1 9627.897,E2 9627.897} C_VEL
LIN {X 0,Y 412.506,Z 793.657,A -85,B 0,C 180,E1 9632.104,E2 9632.104} C_VEL
LIN {X 0,Y 412.704,Z 789.093,A -85,B 0,C 180,E1 9637.912,E2 9637.912} C_VEL
LIN {X 0,Y 413.303,Z 779.919,A -85,B 0,C 180,E1 9643.408,E2 9643.408} C_VEL
LIN {X 0,Y 414.865,Z 766.18,A -85,B 0,C 180,E1 9648.681,E2 9648.681} C_VEL
LIN {X 0,Y 418.034,Z 744.751,A -85,B 0,C 180,E1 9654.421,E2 9654.421} C_VEL
LIN {X 0,Y 422.888,Z 717.779,A -85,B 0,C 180,E1 9659.689,E2 9659.689} C_VEL
LIN {X 0,Y 428.669,Z 686.849,A -85,B 0,C 180,E1 9664.213,E2 9664.213} C_VEL
LIN {X 0,Y 435.366,Z 649.777,A -85,B 0,C 180,E1 9668.279,E2 9668.279} C_VEL
LIN {X 0,Y 441.916,Z 611.13,A -85,B 0,C 180,E1 9671.429,E2 9671.429} C_VEL
LIN {X 0,Y 447.814,Z 569.181,A -85,B 0,C 180,E1 9673.844,E2 9673.844} C_VEL
LIN {X 0,Y 450.771,Z 537.385,A -85,B 0,C 180,E1 9675.145,E2 9675.145} C_VEL
LIN {X 0,Y 434.159,Z 501.294,A -85,B 0,C 180,E1 9678.504,E2 9678.504} C_VEL
LIN {X 0,Y 413.707,Z 468.206,A -85,B 0,C 180,E1 9682.458,E2 9682.458} C_VEL
LIN {X 0,Y 411.184,Z 462.44,A -85,B 0,C 180,E1 9683.146,E2 9683.146} C_VEL
LIN {X 0,Y 411.212,Z 462.44,A -85,B 0,C 180,E1 9688.972,E2 9688.972} C_VEL
LIN {X 0,Y 411.389,Z 462.44,A -85,B 0,C 180,E1 9693.792,E2 9693.792} C_VEL
LIN {X 0,Y 411.672,Z 462.44,A -85,B 0,C 180,E1 9700.67,E2 9700.67} C_VEL
LIN {X 0,Y 411.722,Z 462.44,A -85,B 0,C 180,E1 9707.253,E2 9707.253} C_VEL
LIN {X 0,Y 412.167,Z 462.44,A -85,B 0,C 180,E1 9713.672,E2 9713.672} C_VEL
LIN {X 0,Y 412.394,Z 462.44,A -85,B 0,C 180,E1 9719.999,E2 9719.999} C_VEL
LIN {X 0,Y 412.107,Z 462.44,A -85,B 0,C 180,E1 9726.326,E2 9726.326} C_VEL
LIN {X 0,Y 411.854,Z 462.44,A -85,B 0,C 180,E1 9732.741,E2 9732.741} C_VEL
LIN {X 0,Y 411.625,Z 462.44,A -85,B 0,C 180,E1 9739.329,E2 9739.329} C_VEL
LIN {X 0,Y 411.34,Z 462.44,A -85,B 0,C 180,E1 9746.209,E2 9746.209} C_VEL
LIN {X 0,Y 411.26,Z 462.44,A -85,B 0,C 180,E1 9753.516,E2 9753.516} C_VEL
LIN {X 0,Y 411.113,Z 462.44,A -85,B 0,C 180,E1 9760.941,E2 9760.941} C_VEL
LIN {X 0,Y 411.117,Z 462.44,A -85,B 0,C 180,E1 9761.444,E2 9761.444} C_VEL
LIN {X 0,Y 413.321,Z 467.92,A -85,B 0,C 180,E1 9761.967,E2 9761.967} C_VEL
LIN {X 0,Y 433.441,Z 499.42,A -85,B 0,C 180,E1 9765.786,E2 9765.786} C_VEL
LIN {X 0,Y 450.367,Z 529.706,A -85,B 0,C 180,E1 9768.846,E2 9768.846} C_VEL
LIN {X 0,Y 446.35,Z 571.418,A -85,B 0,C 180,E1 9770.424,E2 9770.424} C_VEL
LIN {X 0,Y 440.62,Z 609.699,A -85,B 0,C 180,E1 9772.724,E2 9772.724} C_VEL
LIN {X 0,Y 434.222,Z 644.18,A -85,B 0,C 180,E1 9775.707,E2 9775.707} C_VEL
LIN {X 0,Y 427.704,Z 675.307,A -85,B 0,C 180,E1 9779.41,E2 9779.41} C_VEL
LIN {X 0,Y 421.828,Z 701.785,A -85,B 0,C 180,E1 9783.656,E2 9783.656} C_VEL
LIN {X 0,Y 417.155,Z 724.989,A -85,B 0,C 180,E1 9788.718,E2 9788.718} C_VEL
LIN {X 0,Y 414.359,Z 742.862,A -85,B 0,C 180,E1 9794.094,E2 9794.094} C_VEL
LIN {X 0,Y 413.119,Z 755.027,A -85,B 0,C 180,E1 9799.441,E2 9799.441} C_VEL
LIN {X 0,Y 412.661,Z 761.082,A -85,B 0,C 180,E1 9803.68,E2 9803.68} C_VEL
LIN {X 0,Y 412.501,Z 764.097,A -85,B 0,C 180,E1 9807.896,E2 9807.896} C_VEL
LIN {X 0,Y 412.612,Z 764.049,A -85,B 0,C 180,E1 9812.103,E2 9812.103} C_VEL
LIN {X 0,Y 412.826,Z 758.865,A -85,B 0,C 180,E1 9818.05,E2 9818.05} C_VEL
LIN {X 0,Y 413.724,Z 748.773,A -85,B 0,C 180,E1 9823.504,E2 9823.504} C_VEL
LIN {X 0,Y 415.704,Z 733.844,A -85,B 0,C 180,E1 9828.76,E2 9828.76} C_VEL
LIN {X 0,Y 419.493,Z 713.185,A -85,B 0,C 180,E1 9833.958,E2 9833.958} C_VEL
LIN {X 0,Y 424.738,Z 688.577,A -85,B 0,C 180,E1 9838.53,E2 9838.53} C_VEL
LIN {X 0,Y 430.895,Z 660.201,A -85,B 0,C 180,E1 9842.441,E2 9842.441} C_VEL
LIN {X 0,Y 437.348,Z 627.963,A -85,B 0,C 180,E1 9845.728,E2 9845.728} C_VEL
LIN {X 0,Y 443.408,Z 592.056,A -85,B 0,C 180,E1 9848.361,E2 9848.361} C_VEL
LIN {X 0,Y 448.36,Z 554.241,A -85,B 0,C 180,E1 9850.224,E2 9850.224} C_VEL
LIN {X 0,Y 450.004,Z 529.361,A -85,B 0,C 180,E1 9851.116,E2 9851.116} C_VEL
LIN {X 0,Y 425.685,Z 486.324,A -85,B 0,C 180,E1 9855.534,E2 9855.534} C_VEL
LIN {X 0,Y 411.373,Z 464.114,A -85,B 0,C 180,E1 9858.355,E2 9858.355} C_VEL
LIN {X 0,Y 411.176,Z 462.44,A -85,B 0,C 180,E1 9858.491,E2 9858.491} C_VEL
LIN {X 0,Y 411.127,Z 462.44,A -85,B 0,C 180,E1 9864.119,E2 9864.119} C_VEL
LIN {X 0,Y 411.329,Z 462.44,A -85,B 0,C 180,E1 9871.415,E2 9871.415} C_VEL
LIN {X 0,Y 411.567,Z 462.44,A -85,B 0,C 180,E1 9878.418,E2 9878.418} C_VEL
LIN {X 0,Y 411.871,Z 462.44,A -85,B 0,C 180,E1 9885.091,E2 9885.091} C_VEL
LIN {X 0,Y 412.079,Z 462.44,A -85,B 0,C 180,E1 9891.551,E2 9891.551} C_VEL
LIN {X 0,Y 412.357,Z 462.44,A -85,B 0,C 180,E1 9897.897,E2 9897.897} C_VEL
LIN {X 0,Y 412.2,Z 462.44,A -85,B 0,C 180,E1 9904.214,E2 9904.214} C_VEL
LIN {X 0,Y 411.916,Z 462.44,A -85,B 0,C 180,E1 9910.591,E2 9910.591} C_VEL
LIN {X 0,Y 411.726,Z 462.44,A -85,B 0,C 180,E1 9917.109,E2 9917.109} C_VEL
LIN {X 0,Y 411.49,Z 462.44,A -85,B 0,C 180,E1 9923.874,E2 9923.874} C_VEL
LIN {X 0,Y 411.347,Z 462.44,A -85,B 0,C 180,E1 9928.586,E2 9928.586} C_VEL
LIN {X 0,Y 411.172,Z 462.44,A -85,B 0,C 180,E1 9936.097,E2 9936.097} C_VEL
LIN {X 0,Y 411.196,Z 462.762,A -85,B 0,C 180,E1 9936.98,E2 9936.98} C_VEL
LIN {X 0,Y 413.668,Z 468.169,A -85,B 0,C 180,E1 9937.547,E2 9937.547} C_VEL
LIN {X 0,Y 434.134,Z 501.303,A -85,B 0,C 180,E1 9941.499,E2 9941.499} C_VEL
LIN {X 0,Y 451.051,Z 537.938,A -85,B 0,C 180,E1 9944.913,E2 9944.913} C_VEL
LIN {X 0,Y 446.581,Z 578.746,A -85,B 0,C 180,E1 9946.631,E2 9946.631} C_VEL
LIN {X 0,Y 440.605,Z 618.69,A -85,B 0,C 180,E1 9949.109,E2 9949.109} C_VEL
LIN {X 0,Y 434.13,Z 656.549,A -85,B 0,C 180,E1 9952.385,E2 9952.385} C_VEL
LIN {X 0,Y 427.804,Z 691.003,A -85,B 0,C 180,E1 9956.331,E2 9956.331} C_VEL
LIN {X 0,Y 422.257,Z 720.849,A -85,B 0,C 180,E1 9960.839,E2 9960.839} C_VEL
LIN {X 0,Y 419.596,Z 735.594,A -85,B 0,C 180,E1 9963.607,E2 9963.607} C_VEL
LIN {X 0,Y 414.181,Z 745.156,A -85,B 0,C 180,E1 9965.489,E2 9965.489} C_VEL
LIN {X 0,Y 408.927,Z 753.833,A -85,B 0,C 180,E1 9967.49,E2 9967.49} C_VEL
LIN {X 0,Y 406.297,Z 772.247,A -85,B 0,C 180,E1 9973.213,E2 9973.213} C_VEL
LIN {X 0,Y 404.988,Z 785.264,A -85,B 0,C 180,E1 9979.226,E2 9979.226} C_VEL
LIN {X 0,Y 404.749,Z 790.904,A -85,B 0,C 180,E1 9983.556,E2 9983.556} C_VEL
LIN {X 0,Y 404.718,Z 793.657,A -85,B 0,C 180,E1 9987.856,E2 9987.856} C_VEL
LIN {X 0,Y 404.614,Z 793.657,A -85,B 0,C 180,E1 9992.145,E2 9992.145} C_VEL
LIN {X 0,Y 404.787,Z 789.402,A -85,B 0,C 180,E1 9997.791,E2 9997.791} C_VEL
LIN {X 0,Y 405.32,Z 781.236,A -85,B 0,C 180,E1 10002.952,E2 10002.952} C_VEL
LIN {X 0,Y 406.98,Z 766.732,A -85,B 0,C 180,E1 10008.718,E2 10008.718} C_VEL
LIN {X 0,Y 410.137,Z 746.276,A -85,B 0,C 180,E1 10014.404,E2 10014.404} C_VEL
LIN {X 0,Y 414.817,Z 721.159,A -85,B 0,C 180,E1 10019.522,E2 10019.522} C_VEL
LIN {X 0,Y 420.635,Z 691.32,A -85,B 0,C 180,E1 10024.123,E2 10024.123} C_VEL
LIN {X 0,Y 427.365,Z 657.098,A -85,B 0,C 180,E1 10028.149,E2 10028.149} C_VEL
LIN {X 0,Y 434.122,Z 620.194,A -85,B 0,C 180,E1 10031.414,E2 10031.414} C_VEL
LIN {X 0,Y 440.252,Z 581.603,A -85,B 0,C 180,E1 10033.885,E2 10033.885} C_VEL
LIN {X 0,Y 444.547,Z 540.264,A -85,B 0,C 180,E1 10035.759,E2 10035.759} C_VEL
LIN {X 0,Y 429.362,Z 506.279,A -85,B 0,C 180,E1 10039.025,E2 10039.025} C_VEL
LIN {X 0,Y 409.815,Z 474.256,A -85,B 0,C 180,E1 10042.941,E2 10042.941} C_VEL
LIN {X 0,Y 403.435,Z 464.142,A -85,B 0,C 180,E1 10044.358,E2 10044.358} C_VEL
